(* Logix 5000 project; controller R1USB70001_CWRU_LOAD_20111116 vendor 1 type 14 code 54 rev 19.11; software revision 19.01 *)

TASK MainTask (continuous, watchdog 500 ms) : MainProgram

MODULES
   Local : vendor 1 type 14 code 54 (ICP 2, rev 19.11)
      CNB_LOAD : vendor 1 type 12 code 21 (ICP 0, rev 20.1)
         ACNR_RP_SC_N4 : vendor 1 type 12 code 111 (ControlNet 4, rev 1.1, Output RPI 8 ms)
            IE4C_RP_SC_S1 : 1734-IE4C (PointIO 1, rev 3.1, Input RPI 8 ms)
            IE4C_RP_SC_S2 : 1734-IE4C (PointIO 2, rev 3.1, Input RPI 8 ms)
            IE4C_RP_SC_S4 : 1734-IE4C (PointIO 4, rev 3.1, Input RPI 8 ms)
            IE4C_RP_SC_S3 : 1734-IE4C (PointIO 3, rev 3.1, Input RPI 8 ms)
            IE4C_RP_SC_S5 : 1734-IE4C (PointIO 5, rev 3.1, Input RPI 8 ms)
            IE4C_RP_SC_S6 : 1734-IE4C (PointIO 6, rev 3.1, Input RPI 8 ms)
            IE4C_RP_SC_S7 : 1734-IE4C (PointIO 7, rev 3.1, Input RPI 8 ms)
            IB8_RP_SC_S8 : 1734-IB8 (PointIO 8, rev 3.1)
            OB8_RP_SC_S10 : 1734-OB8 (PointIO 10, rev 3.1)
            OB8_RP_SC_S11 : 1734-OB8 (PointIO 11, rev 3.1)
            OB8_RP_SC_S12 : 1734-OB8 (PointIO 12, rev 3.1)
            OB8_RP_SC_S9 : 1734-OB8 (PointIO 9, rev 3.1)
         ACNR_CP_SC_N5 : vendor 1 type 12 code 111 (ControlNet 5, rev 1.1, Output RPI 8 ms)
            IE4C_CP_SC_S8 : 1734-IE4C (PointIO 8, rev 3.1, Input RPI 8 ms)
            IE4C_CP_SC_S1 : 1734-IE4C (PointIO 1, rev 3.1, Input RPI 8 ms)
            IE4C_CP_SC_S2 : 1734-IE4C (PointIO 2, rev 3.1, Input RPI 8 ms)
            IE4C_CP_SC_S3 : 1734-IE4C (PointIO 3, rev 3.1, Input RPI 8 ms)
            IE4C_CP_SC_S4 : 1734-IE4C (PointIO 4, rev 3.1, Input RPI 8 ms)
            IE4C_CP_SC_S6 : 1734-IE4C (PointIO 6, rev 3.1, Input RPI 8 ms)
            IE4C_CP_SC_S5 : 1734-IE4C (PointIO 5, rev 3.1, Input RPI 8 ms)
            IE4C_CP_SC_S7 : 1734-IE4C (PointIO 7, rev 3.1, Input RPI 8 ms)
            IB8_CP_SC_S9 : 1734-IB8 (PointIO 9, rev 3.1)
            OB8_CP_SC_S14 : 1734-OB8 (PointIO 13, rev 3.1)
            OB8_CP_SC_S13 : 1734-OB8 (PointIO 12, rev 3.1)
            OB8_CP_SC_S11 : 1734-OB8 (PointIO 10, rev 3.1)
            OB8_CP_SC_S12 : 1734-OB8 (PointIO 11, rev 3.1)
      EN2T_LOAD : 1756-EN2T (ICP 1, Ethernet 10.88.0.104, rev 4.3)
END_MODULES

VAR_GLOBAL   (* controller tags *)
   CL_LP_B1_ACAM : ALIAS FOR ACNR_CP_SC_N5:1:I.Ch1Data;
   CL_LP_B1_ACVS : ALIAS FOR ACNR_CP_SC_N5:9:I.1;
   CL_LP_B1_L1_ACAM : ALIAS FOR ACNR_CP_SC_N5:1:I.Ch2Data;
   CL_LP_B1_L2_ACAM : ALIAS FOR ACNR_CP_SC_N5:1:I.Ch3Data;
   CL_LP_B1_L3_ACAM : ALIAS FOR ACNR_CP_SC_N5:2:I.Ch0Data;
   CL_LP_B1_L4_ACAM : ALIAS FOR ACNR_CP_SC_N5:2:I.Ch1Data;
   CL_LP_B1_L5_ACAM : ALIAS FOR ACNR_CP_SC_N5:2:I.Ch2Data;
   CL_LP_B2_ACAM : ALIAS FOR ACNR_CP_SC_N5:2:I.Ch3Data;
   CL_LP_B2_ACVS : ALIAS FOR ACNR_CP_SC_N5:9:I.2;
   CL_LP_B2_L1_ACAM : ALIAS FOR ACNR_CP_SC_N5:3:I.Ch0Data;
   CL_LP_B2_L2_ACAM : ALIAS FOR ACNR_CP_SC_N5:3:I.Ch1Data;
   CL_LP_B2_L3_ACAM : ALIAS FOR ACNR_CP_SC_N5:3:I.Ch2Data;
   CL_LP_B2_L4_ACAM : ALIAS FOR ACNR_CP_SC_N5:3:I.Ch3Data;
   CL_LP_B2_L5_ACAM : ALIAS FOR ACNR_CP_SC_N5:4:I.Ch0Data;
   CL_LP_ML_ACAM : ALIAS FOR ACNR_CP_SC_N5:1:I.Ch0Data;
   CL_LP_ML_ACVT : ALIAS FOR ACNR_CP_SC_N5:7:I.Ch2Data;
   CL_TIMER00 : TIMER;
   COM_B1_Alias : ALIAS FOR ACNR_CP_SC_N5:10:O.1;
   COM_B1_LOAD1_Alias : ALIAS FOR ACNR_CP_SC_N5:10:O.2;
   COM_B1_LOAD1_USER : BOOL;
   COM_B1_LOAD2_Alias : ALIAS FOR ACNR_CP_SC_N5:10:O.3;
   COM_B1_LOAD2_USER : BOOL;
   COM_B1_LOAD3_Alias : ALIAS FOR ACNR_CP_SC_N5:10:O.4;
   COM_B1_LOAD3_USER : BOOL;
   COM_B1_LOAD4_Alias : ALIAS FOR ACNR_CP_SC_N5:10:O.5;
   COM_B1_LOAD4_USER : BOOL;
   COM_B1_LOAD5_Alias : ALIAS FOR ACNR_CP_SC_N5:10:O.6;
   COM_B1_LOAD5_USER : BOOL;
   COM_B1_USER : BOOL;
   COM_B2_Alias : ALIAS FOR ACNR_CP_SC_N5:10:O.7;
   COM_B2_LOAD1_Alias : ALIAS FOR ACNR_CP_SC_N5:11:O.0;
   COM_B2_LOAD1_USER : BOOL;
   COM_B2_LOAD2_Alias : ALIAS FOR ACNR_CP_SC_N5:11:O.1;
   COM_B2_LOAD2_USER : BOOL;
   COM_B2_LOAD3_Alias : ALIAS FOR ACNR_CP_SC_N5:11:O.2;
   COM_B2_LOAD3_USER : BOOL;
   COM_B2_LOAD4_Alias : ALIAS FOR ACNR_CP_SC_N5:11:O.3;
   COM_B2_LOAD4_USER : BOOL;
   COM_B2_LOAD5_Alias : ALIAS FOR ACNR_CP_SC_N5:11:O.4;
   COM_B2_LOAD5_USER : BOOL;
   COM_B2_USER : BOOL;
   COM_MAIN_Alias : ALIAS FOR ACNR_CP_SC_N5:10:O.0;
   COM_MAIN_CLOSE : BOOL;
   COM_MAIN_CLOSE_Alias : BOOL;
   COM_MAIN_USER : BOOL;
   Comment : DINT[2] := ([0] := 3);
   HMI_Intfc_Read_Buffer : DINT[66] := ([0] := 235, [1] := 560, [2] := 5614, [3] := -31, [4] := -66, [5] := -101, [6] := 317, [7] := -1, [8] := 114, [9] := 102, [10] := 69, [11] := -7, [12] := 37, [13] := -1, [14] := 64, [15] := 82, [16] := -48, [17] := 42, [18] := 138, [20] := 25, [21] := 35, [22] := -29, [23] := 66, [25] := 7, [26] := -17, [27] := -13, [28] := 22, [29] := 1048839, [30] := 430, [31] := 431, [34] := 97, [35] := -66, [36] := -44, [37] := 52, [38] := 59, [40] := 5, [41] := 5, [42] := 68, [43] := 24, [44] := -84, [46] := -1, [47] := 56, [48] := -6, [49] := 66, [50] := 126, [51] := 109, [53] := 64, [54] := 77, [55] := 6, [56] := 31, [57] := 37, [59] := 1, [60] := 3294, [61] := -16, [62] := -15, [63] := -12);
        [0]   // RL_LP_ML_ACAM
        [1]   // RL_LP_B1_ACAM
        [2]   // RL_LP_B1_L1_ACAM
        [3]   // RL_LP_B1_L2_ACAM
        [4]   // RL_LP_B1_L3_ACAM
        [5]   // RL_LP_B1_L4_ACAM
        [6]   // RL_LP_B1_L5_ACAM
        [7]   // RL_LP_B2_ACAM
        [8]   // RL_LP_B2_L1_ACAM
        [9]   // RL_LP_B2_L2_ACAM
        [10]   // RL_LP_B2_L3_ACAM
        [11]   // RL_LP_B2_L4_ACAM
        [26]   // SPARE RESERVED FOR SLOT 7 CHANNEL 2
        [27]   // SPARE RESERVED FOR SLOT 7 CHANNEL 3
        [63]   // SPARE RESERVED FOR SLOT 8 CHANNEL 3
        [62]   // SPARE RESERVED FOR SLOT 8 CHANNEL 2
        [61]   // SPARE RESERVED FOR SLOT 8 CHANNEL 1
        [60]   // SPARE RESERVED FOR SLOT 8 CHANNEL 0
        [12]   // RL_LP_B2_L5_ACAM
        [13]   // RL_LP_B3_ACAM
        [14]   // RL_LP_B3_L1_ACAM
        [15]   // RL_LP_B3_L2_ACAM
        [16]   // RL_LP_B3_L3_ACAM
        [17]   // RL_LP_B3_L4_ACAM
        [18]   // RL_LP_B3_L5_ACAM
        [19]   // RL_LP_B4_ACAM
        [20]   // RL_LP_B4_L1_ACAM
        [21]   // RL_LP_B4_L2_ACAM
        [22]   // RL_LP_B4_L3_ACAM
        [23]   // RL_LP_B4_L4_ACAM
        [24]   // RL_LP_B4_L5_ACAM
        [25]   // RL_LP_ML_ACVT
        [28].1   // RL_LP_B1_ACVS
        [28].2   // RL_LP_B2_ACVS
        [28].3   // RL_LP_B3_ACVS
        [28].4   // RL_LP_B4_ACVS
        [29].0   // RL_LP_ML_CS
        [29].1   // RL_LP_B1_CS
        [29].2   // RL_LP_B1_L1_CS
        [29].3   // RL_LP_B1_L2_CS
        [29].4   // RL_LP_B1_L3_CS
        [29].5   // RL_LP_B1_L4_CS
        [29].6   // RL_LP_B1_L5_CS
        [29].8   // RL_LP_B2_CS
        [29].9   // RL_LP_B2_L1_CS
        [29].10   // RL_LP_B2_L2_CS
        [29].11   // RL_LP_B2_L3_CS
        [29].12   // RL_LP_B2_L4_CS
        [29].13   // RL_LP_B2_L5_CS
        [29].14   // RL_LP_B3_CS
        [29].15   // RL_LP_B3_L1_CS
        [29].16   // RL_LP_B3_L2_CS
        [29].17   // RL_LP_B3_L3_CS
        [29].18   // RL_LP_B3_L4_CS
        [29].19   // RL_LP_B3_L5_CS
        [29].20   // RL_LP_B4_CS
        [29].21   // RL_LP_B4_L1_CS
        [29].22   // RL_LP_B4_L2_CS
        [29].23   // RL_LP_B4_L3_CS
        [29].24   // RL_LP_B4_L4_CS
        [29].25   // RL_LP_B4_L5_CS
        [32]   // CL_LP_ML_ACAM
        [33]   // CL_LP_B1_ACAM
        [34]   // CL_LP_B1_L1_ACAM
        [35]   // CL_LP_B1_L2_ACAM
        [36]   // CL_LP_B1_L3_ACAM
        [37]   // CL_LP_B1_L4_ACAM
        [38]   // CL_LP_B1_L5_ACAM
        [39]   // CL_LP_B2_ACAM
        [40]   // CL_LP_B2_L1_ACAM
        [41]   // CL_LP_B2_L2_ACAM
        [42]   // CL_LP_B2_L3_ACAM
        [43]   // CL_LP_B2_L4_ACAM
        [44]   // CL_LP_B2_L5_ACAM
        [45]   // IL_LP_ML_ACAM
        [46]   // IL_LP_B1_ACAM
        [47]   // IL_LP_B1_L1_ACAM
        [48]   // IL_LP_B1_L2_ACAM
        [49]   // IL_LP_B1_L3_ACAM
        [50]   // IL_LP_B1_L4_ACAM
        [51]   // IL_LP_B1_L5_ACAM
        [52]   // IL_LP_B2_ACAM
        [53]   // IL_LP_B2_L1_ACAM
        [54]   // IL_LP_B2_L2_ACAM
        [55]   // IL_LP_B2_L3_ACAM
        [56]   // IL_LP_B2_L4_ACAM
        [57]   // IL_LP_B2_L5_ACAM
        [58]   // CL_LP_ML_ACVT
        [59]   // IL_LP_ML_ACVT
        [64].1   // CL_LP_B1_ACVS
        [64].2   // CL_LP_B2_ACVS
        [64].4   // IL_LP_B1_ACVS
        [64].5   // IL_LP_B2_ACVS
        [65].0   // CL_LP_ML_CS
        [65].1   // CL_LP_B1_CS
        [65].2   // CL_LP_B1_L1_CS
        [65].3   // CL_LP_B1_L2_CS
        [65].4   // CL_LP_B1_L3_CS
        [65].5   // CL_LP_B1_L4_CS
        [65].6   // CL_LP_B1_L5_CS
        [65].7   // CL_LP_B2_CS
        [65].8   // CL_LP_B2_L1_CS
        [65].9   // CL_LP_B2_L2_CS
        [65].10   // CL_LP_B2_L3_CS
        [65].11   // CL_LP_B2_L4_CS
        [65].12   // CL_LP_B2_L5_CS
        [65].13   // IL_LP_ML_CS
        [65].14   // IL_LP_B1_CS
        [65].15   // IL_LP_B1_L1_CS
        [65].16   // IL_LP_B1_L2_CS
        [65].17   // IL_LP_B1_L3_CS
        [65].18   // IL_LP_B1_L4_CS
        [65].19   // IL_LP_B1_L5_CS
        [65].20   // IL_LP_B2_CS
        [65].21   // IL_LP_B2_L1_CS
        [65].22   // IL_LP_B2_L2_CS
        [65].23   // IL_LP_B2_L3_CS
        [65].24   // IL_LP_B2_L4_CS
        [65].25   // IL_LP_B2_L5_CS
   IL_LP_B1_ACAM : ALIAS FOR ACNR_CP_SC_N5:4:I.Ch2Data;
   IL_LP_B1_ACVS : ALIAS FOR ACNR_CP_SC_N5:9:I.4;
   IL_LP_B1_L1_ACAM : ALIAS FOR ACNR_CP_SC_N5:4:I.Ch3Data;
   IL_LP_B1_L2_ACAM : ALIAS FOR ACNR_CP_SC_N5:5:I.Ch0Data;
   IL_LP_B1_L3_ACAM : ALIAS FOR ACNR_CP_SC_N5:5:I.Ch1Data;
   IL_LP_B1_L4_ACAM : ALIAS FOR ACNR_CP_SC_N5:5:I.Ch2Data;
   IL_LP_B1_L5_ACAM : ALIAS FOR ACNR_CP_SC_N5:5:I.Ch3Data;
   IL_LP_B2_ACAM : ALIAS FOR ACNR_CP_SC_N5:6:I.Ch0Data;
   IL_LP_B2_ACVS : ALIAS FOR ACNR_CP_SC_N5:9:I.5;
   IL_LP_B2_L1_ACAM : ALIAS FOR ACNR_CP_SC_N5:6:I.Ch1Data;
   IL_LP_B2_L2_ACAM : ALIAS FOR ACNR_CP_SC_N5:6:I.Ch2Data;
   IL_LP_B2_L3_ACAM : ALIAS FOR ACNR_CP_SC_N5:6:I.Ch3Data;
   IL_LP_B2_L4_ACAM : ALIAS FOR ACNR_CP_SC_N5:7:I.Ch0Data;
   IL_LP_B2_L5_ACAM : ALIAS FOR ACNR_CP_SC_N5:7:I.Ch1Data;
   IL_LP_ML_ACAM : ALIAS FOR ACNR_CP_SC_N5:4:I.Ch1Data;
   IL_LP_ML_ACVT : ALIAS FOR ACNR_CP_SC_N5:7:I.Ch3Data;
   IND_B1_Alias : ALIAS FOR ACNR_CP_SC_N5:11:O.6;
   IND_B1_LOAD1_Alias : ALIAS FOR ACNR_CP_SC_N5:11:O.7;
   IND_B1_LOAD1_USER : BOOL;
   IND_B1_LOAD2_Alias : ALIAS FOR ACNR_CP_SC_N5:12:O.0;
   IND_B1_LOAD2_USER : BOOL;
   IND_B1_LOAD3_Alias : ALIAS FOR ACNR_CP_SC_N5:12:O.1;
   IND_B1_LOAD3_USER : BOOL;
   IND_B1_LOAD4_Alias : ALIAS FOR ACNR_CP_SC_N5:12:O.2;
   IND_B1_LOAD4_USER : BOOL;
   IND_B1_LOAD5_Alias : ALIAS FOR ACNR_CP_SC_N5:12:O.3;
   IND_B1_LOAD5_USER : BOOL;
   IND_B1_USER : BOOL;
   IND_B2_Alias : ALIAS FOR ACNR_CP_SC_N5:12:O.4;
   IND_B2_LOAD1_Alias : ALIAS FOR ACNR_CP_SC_N5:12:O.5;
   IND_B2_LOAD1_USER : BOOL;
   IND_B2_LOAD2_Alias : ALIAS FOR ACNR_CP_SC_N5:12:O.6;
   IND_B2_LOAD2_USER : BOOL;
   IND_B2_LOAD3_Alias : ALIAS FOR ACNR_CP_SC_N5:12:O.7;
   IND_B2_LOAD3_USER : BOOL;
   IND_B2_LOAD4_Alias : ALIAS FOR ACNR_CP_SC_N5:13:O.0;
   IND_B2_LOAD4_USER : BOOL;
   IND_B2_LOAD5_Alias : ALIAS FOR ACNR_CP_SC_N5:13:O.1;
   IND_B2_LOAD5_USER : BOOL;
   IND_B2_USER : BOOL;
   IND_MAIN_Alias : ALIAS FOR ACNR_CP_SC_N5:11:O.5;
   IND_MAIN_USER : BOOL;
   RES_B1_Alias : ALIAS FOR ACNR_RP_SC_N4:9:O.1;
   RES_B1_LOAD1_Alias : ALIAS FOR ACNR_RP_SC_N4:9:O.2;
   RES_B1_LOAD1_USER : BOOL;
   RES_B1_LOAD2_Alias : ALIAS FOR ACNR_RP_SC_N4:9:O.3;
   RES_B1_LOAD2_USER : BOOL;
   RES_B1_LOAD3_Alias : ALIAS FOR ACNR_RP_SC_N4:9:O.4;
   RES_B1_LOAD3_USER : BOOL;
   RES_B1_LOAD4_Alias : ALIAS FOR ACNR_RP_SC_N4:9:O.5;
   RES_B1_LOAD4_USER : BOOL;
   RES_B1_LOAD5_Alias : ALIAS FOR ACNR_RP_SC_N4:9:O.6;
   RES_B1_LOAD5_USER : BOOL;
   RES_B1_USER : BOOL;
   RES_B2_Alias : ALIAS FOR ACNR_RP_SC_N4:10:O.0;
   RES_B2_LOAD1_Alias : ALIAS FOR ACNR_RP_SC_N4:10:O.1;
   RES_B2_LOAD1_USER : BOOL;
   RES_B2_LOAD2_Alias : ALIAS FOR ACNR_RP_SC_N4:10:O.2;
   RES_B2_LOAD2_USER : BOOL;
   RES_B2_LOAD3_Alias : ALIAS FOR ACNR_RP_SC_N4:10:O.3;
   RES_B2_LOAD3_USER : BOOL;
   RES_B2_LOAD4_Alias : ALIAS FOR ACNR_RP_SC_N4:10:O.4;
   RES_B2_LOAD4_USER : BOOL;
   RES_B2_LOAD5_Alias : ALIAS FOR ACNR_RP_SC_N4:10:O.5;
   RES_B2_LOAD5_USER : BOOL;
   RES_B2_USER : BOOL;
   RES_B3_Alias : ALIAS FOR ACNR_RP_SC_N4:10:O.6;
   RES_B3_LOAD1_Alias : ALIAS FOR ACNR_RP_SC_N4:10:O.7;
   RES_B3_LOAD1_USER : BOOL;
   RES_B3_LOAD2_Alias : ALIAS FOR ACNR_RP_SC_N4:11:O.0;
   RES_B3_LOAD2_USER : BOOL;
   RES_B3_LOAD3_Alias : ALIAS FOR ACNR_RP_SC_N4:11:O.1;
   RES_B3_LOAD3_USER : BOOL;
   RES_B3_LOAD4_Alias : ALIAS FOR ACNR_RP_SC_N4:11:O.2;
   RES_B3_LOAD4_USER : BOOL;
   RES_B3_LOAD5_Alias : ALIAS FOR ACNR_RP_SC_N4:11:O.3;
   RES_B3_LOAD5_USER : BOOL;
   RES_B3_USER : BOOL;
   RES_B4_Alias : ALIAS FOR ACNR_RP_SC_N4:11:O.4;
   RES_B4_LOAD1_Alias : ALIAS FOR ACNR_RP_SC_N4:11:O.5;
   RES_B4_LOAD1_USER : BOOL;
   RES_B4_LOAD2_Alias : ALIAS FOR ACNR_RP_SC_N4:11:O.6;
   RES_B4_LOAD2_USER : BOOL;
   RES_B4_LOAD3_Alias : ALIAS FOR ACNR_RP_SC_N4:11:O.7;
   RES_B4_LOAD3_USER : BOOL;
   RES_B4_LOAD4_Alias : ALIAS FOR ACNR_RP_SC_N4:12:O.0;
   RES_B4_LOAD4_USER : BOOL;
   RES_B4_LOAD5_Alias : ALIAS FOR ACNR_RP_SC_N4:12:O.1;
   RES_B4_LOAD5_USER : BOOL;
   RES_B4_USER : BOOL;
   RES_MAIN_Alias : ALIAS FOR ACNR_RP_SC_N4:9:O.0;
   RES_MAIN_USER : BOOL;
   RESB1_LOAD1_USER : BOOL;
   RESB2_LOAD2_USER : BOOL;
   RL_LP_B1_ACAM : ALIAS FOR ACNR_RP_SC_N4:1:I.Ch1Data;
   RL_LP_B1_ACVS : ALIAS FOR ACNR_RP_SC_N4:8:I.1;
   RL_LP_B1_L1_ACAM : ALIAS FOR ACNR_RP_SC_N4:1:I.Ch2Data;
   RL_LP_B1_L2_ACAM : ALIAS FOR ACNR_RP_SC_N4:1:I.Ch3Data;
   RL_LP_B1_L3_ACAM : ALIAS FOR ACNR_RP_SC_N4:2:I.Ch0Data;
   RL_LP_B1_L4_ACAM : ALIAS FOR ACNR_RP_SC_N4:2:I.Ch1Data;
   RL_LP_B1_L5_ACAM : ALIAS FOR ACNR_RP_SC_N4:2:I.Ch2Data;
   RL_LP_B2_ACAM : ALIAS FOR ACNR_RP_SC_N4:2:I.Ch3Data;
   RL_LP_B2_ACVS : ALIAS FOR ACNR_RP_SC_N4:8:I.2;
   RL_LP_B2_L1_ACAM : ALIAS FOR ACNR_RP_SC_N4:3:I.Ch0Data;
   RL_LP_B2_L2_ACAM : ALIAS FOR ACNR_RP_SC_N4:3:I.Ch1Data;
   RL_LP_B2_L3_ACAM : ALIAS FOR ACNR_RP_SC_N4:3:I.Ch2Data;
   RL_LP_B2_L4_ACAM : ALIAS FOR ACNR_RP_SC_N4:3:I.Ch3Data;
   RL_LP_B2_L5_ACAM : ALIAS FOR ACNR_RP_SC_N4:4:I.Ch0Data;
   RL_LP_B3_ACAM : ALIAS FOR ACNR_RP_SC_N4:4:I.Ch1Data;
   RL_LP_B3_ACVS : ALIAS FOR ACNR_RP_SC_N4:8:I.3;
   RL_LP_B3_L1_ACAM : ALIAS FOR ACNR_RP_SC_N4:4:I.Ch2Data;
   RL_LP_B3_L2_ACAM : ALIAS FOR ACNR_RP_SC_N4:4:I.Ch3Data;
   RL_LP_B3_L3_ACAM : ALIAS FOR ACNR_RP_SC_N4:5:I.Ch0Data;
   RL_LP_B3_L4_ACAM : ALIAS FOR ACNR_RP_SC_N4:5:I.Ch1Data;
   RL_LP_B3_L5_ACAM : ALIAS FOR ACNR_RP_SC_N4:5:I.Ch2Data;
   RL_LP_B4_ACAM : ALIAS FOR ACNR_RP_SC_N4:5:I.Ch3Data;
   RL_LP_B4_ACVS : ALIAS FOR ACNR_RP_SC_N4:8:I.4;
   RL_LP_B4_L1_ACAM : ALIAS FOR ACNR_RP_SC_N4:6:I.Ch0Data;
   RL_LP_B4_L2_ACAM : ALIAS FOR ACNR_RP_SC_N4:6:I.Ch1Data;
   RL_LP_B4_L3_ACAM : ALIAS FOR ACNR_RP_SC_N4:6:I.Ch2Data;
   RL_LP_B4_L4_ACAM : ALIAS FOR ACNR_RP_SC_N4:6:I.Ch3Data;
   RL_LP_B4_L5_ACAM : ALIAS FOR ACNR_RP_SC_N4:7:I.Ch0Data;
   RL_LP_ML_ACAM : ALIAS FOR ACNR_RP_SC_N4:1:I.Ch0Data;
   RL_LP_ML_ACVT : ALIAS FOR ACNR_RP_SC_N4:7:I.Ch1Data;
END_VAR

PROGRAM MainProgram   (* main routine MainRoutine *)
VAR
   COM_B1_CLOSE_PROXY : BOOL;
   COM_B1_CLOSED : BOOL;
   COM_B1_COMMAND_CHANGED : BOOL;
   COM_B1_COMMAND_CHANGED_TIMER : TIMER;
   COM_B1_CURRENT_CHECK : REAL := 0.0059203943;
   COM_B1_CURRENT_RAW : REAL;
   COM_B1_DISCREPANCY : REAL := 0.0059203943;
   COM_B1_FAULT_CANCEL : BOOL := 1;
   COM_B1_FAULT_PENDING : BOOL;
   COM_B1_FAULT_REQ : BOOL;
   COM_B1_FAULT_RETHROW_TIMER : TIMER := (PRE := 100);
   COM_B1_FAULT_TRIP : BOOL;
   COM_B1_INT_REQ_CLOSE : BOOL;
   COM_B1_INT_REQ_CONNECT : BOOL;
   COM_B1_MISMATCH : BOOL;
   COM_B1_NEW_FAULT : BOOL;
   COM_B1_RECLOSE_COUNTER : DINT;
   COM_B1_RECLOSE_OFF : BOOL;
   COM_B1_RECLOSE_TIMER : TIMER := (PRE := 1000);
   COM_B1_RECLOSED : BOOL;
   COM_B1_REQ_CLOSE : BOOL;
   COM_B1_REQ_CONNECT : BOOL;
   COM_B1_REQ_DISCONNECT : BOOL;
   COM_B1_REQ_OPEN : BOOL := 1;
   COM_B1_REQ_RECLOSE : BOOL;
   COM_B1_SENSOR_ERROR : BOOL;
   COM_B1L1_CURRENT : REAL := 0.005920395;
   COM_B1L1_CURRENT_RAW : REAL := 97.0;
   COM_B1L2_CURRENT : REAL := -0.00402831;
   COM_B1L2_CURRENT_RAW : REAL := -66.0;
   COM_B1L3_CURRENT : REAL := -0.002746575;
   COM_B1L3_CURRENT_RAW : REAL := -45.0;
   COM_B1L4_CURRENT : REAL := 0.00317382;
   COM_B1L4_CURRENT_RAW : REAL := 52.0;
   COM_B1L5_CURRENT : REAL := 0.003601065;
   COM_B1L5_CURRENT_RAW : REAL := 59.0;
   COM_B2_CLOSE_PROXY : BOOL;
   COM_B2_CLOSED : BOOL;
   COM_B2_COMMAND_CHANGED : BOOL;
   COM_B2_COMMAND_CHANGED_TIMER : TIMER;
   COM_B2_CURRENT_CHECK : REAL := 0.00109863;
   COM_B2_CURRENT_RAW : REAL;
   COM_B2_DISCREPANCY : REAL := 0.00109863;
   COM_B2_FAULT_CANCEL : BOOL := 1;
   COM_B2_FAULT_PENDING : BOOL;
   COM_B2_FAULT_REQ : BOOL;
   COM_B2_FAULT_RETHROW_TIMER : TIMER := (PRE := 100);
   COM_B2_FAULT_TRIP : BOOL;
   COM_B2_INT_REQ_CLOSE : BOOL;
   COM_B2_INT_REQ_CONNECT : BOOL;
   COM_B2_MISMATCH : BOOL;
   COM_B2_NEW_FAULT : BOOL;
   COM_B2_RECLOSE_COUNTER : DINT;
   COM_B2_RECLOSE_OFF : BOOL;
   COM_B2_RECLOSE_TIMER : TIMER := (PRE := 1000);
   COM_B2_RECLOSED : BOOL;
   COM_B2_REQ_CLOSE : BOOL;
   COM_B2_REQ_CONNECT : BOOL;
   COM_B2_REQ_DISCONNECT : BOOL;
   COM_B2_REQ_OPEN : BOOL := 1;
   COM_B2_REQ_RECLOSE : BOOL;
   COM_B2_SENSOR_ERROR : BOOL;
   COM_B2L1_CURRENT : REAL := 0.000305175;
   COM_B2L1_CURRENT_RAW : REAL := 5.0;
   COM_B2L2_CURRENT : REAL := 0.000305175;
   COM_B2L2_CURRENT_RAW : REAL := 5.0;
   COM_B2L3_CURRENT : REAL := 0.00415038;
   COM_B2L3_CURRENT_RAW : REAL := 68.0;
   COM_B2L4_CURRENT : REAL := 0.00146484;
   COM_B2L4_CURRENT_RAW : REAL := 24.0;
   COM_B2L5_CURRENT : REAL := -0.00512694;
   COM_B2L5_CURRENT_RAW : REAL := -84.0;
   COM_BUS1_CURRENT : REAL;
   COM_BUS2_CURRENT : REAL;
   COM_BUS_FAULT_THRESHOLD : REAL := 2.0;
   COM_HighVoltage : BOOL;
   COM_HighVoltageThreshold : REAL;
   COM_LowVoltage : BOOL;
   COM_LowVoltageThreshold : REAL;
   COM_MAIN_CLOSE_PROXY : BOOL;
   COM_MAIN_CLOSED : BOOL;
   COM_MAIN_COMMAND_CHANGED : BOOL;
   COM_MAIN_COMMAND_CHANGED_TIMER : TIMER;
   COM_MAIN_CURRENT : REAL;
   COM_MAIN_CURRENT_CHECK : REAL;
   COM_MAIN_CURRENT_RAW : REAL;
   COM_MAIN_DISCREPANCY : REAL;
   COM_MAIN_FAULT_CANCEL : BOOL;
   COM_MAIN_FAULT_PENDING : BOOL := 1;
   COM_MAIN_FAULT_REQ : BOOL := 1;
   COM_MAIN_FAULT_RETHROW_TIMER : TIMER := (PRE := 100);
   COM_MAIN_FAULT_THRESHOLD : REAL;
   COM_MAIN_FAULT_TRIP : BOOL := 1;
   COM_MAIN_INT_REQ_CLOSE : BOOL;
   COM_MAIN_INT_REQ_CONNECT : BOOL;
   COM_MAIN_MISMATCH : BOOL := 1;
   COM_MAIN_NEW_FAULT : BOOL;
   COM_MAIN_RECLOSE_COUNTER : DINT := 75;
   COM_MAIN_RECLOSE_OFF : BOOL := 1;
   COM_MAIN_RECLOSE_TIMER : TIMER := (PRE := 1000);
   COM_MAIN_RECLOSED : BOOL;
   COM_MAIN_REQ_CLOSE : BOOL;
   COM_MAIN_REQ_CONNECT : BOOL;
   COM_MAIN_REQ_DISCONNECT : BOOL;
   COM_MAIN_REQ_OPEN : BOOL := 1;
   COM_MAIN_REQ_RECLOSE : BOOL;
   COM_MAIN_SENSOR_ERROR : BOOL;
   COM_MAIN_VOLTAGE : REAL;
   COM_MAIN_VOLTAGE_RAW : REAL;
   CURRENT_SCALE_HIGH : REAL := 0.00061037;
   CURRENT_SCALE_LOW : REAL := 6.1035e-05;
   IND_B1_CLOSE_PROXY : BOOL;
   IND_B1_CLOSED : BOOL;
   IND_B1_COMMAND_CHANGED : BOOL;
   IND_B1_COMMAND_CHANGED_TIMER : TIMER;
   IND_B1_CURRENT_CHECK : REAL := 0.021423286;
   IND_B1_CURRENT_RAW : REAL := -1.0;
   IND_B1_DISCREPANCY : REAL := 0.022033656;
   IND_B1_FAULT_CANCEL : BOOL;
   IND_B1_FAULT_PENDING : BOOL := 1;
   IND_B1_FAULT_REQ : BOOL := 1;
   IND_B1_FAULT_RETHROW_TIMER : TIMER := (PRE := 100);
   IND_B1_FAULT_TRIP : BOOL := 1;
   IND_B1_INT_REQ_CLOSE : BOOL;
   IND_B1_INT_REQ_CONNECT : BOOL;
   IND_B1_MISMATCH : BOOL := 1;
   IND_B1_NEW_FAULT : BOOL;
   IND_B1_RECLOSE_COUNTER : DINT := 75;
   IND_B1_RECLOSE_OFF : BOOL := 1;
   IND_B1_RECLOSE_TIMER : TIMER := (PRE := 1000);
   IND_B1_RECLOSED : BOOL;
   IND_B1_REQ_CLOSE : BOOL;
   IND_B1_REQ_CONNECT : BOOL;
   IND_B1_REQ_DISCONNECT : BOOL;
   IND_B1_REQ_OPEN : BOOL := 1;
   IND_B1_REQ_RECLOSE : BOOL;
   IND_B1_SENSOR_ERROR : BOOL;
   IND_B1L1_CURRENT : REAL := 0.003478995;
   IND_B1L1_CURRENT_RAW : REAL := 57.0;
   IND_B1L2_CURRENT : REAL := -0.00036621;
   IND_B1L2_CURRENT_RAW : REAL := -6.0;
   IND_B1L3_CURRENT : REAL := 0.00402831;
   IND_B1L3_CURRENT_RAW : REAL := 66.0;
   IND_B1L4_CURRENT : REAL := 0.00769041;
   IND_B1L4_CURRENT_RAW : REAL := 126.0;
   IND_B1L5_CURRENT : REAL := 0.00659178;
   IND_B1L5_CURRENT_RAW : REAL := 108.0;
   IND_B2_CLOSE_PROXY : BOOL;
   IND_B2_CLOSED : BOOL;
   IND_B2_COMMAND_CHANGED : BOOL;
   IND_B2_COMMAND_CHANGED_TIMER : TIMER;
   IND_B2_CURRENT_CHECK : REAL := 0.01318356;
   IND_B2_CURRENT_RAW : REAL := -1.0;
   IND_B2_DISCREPANCY : REAL := 0.01379393;
   IND_B2_FAULT_CANCEL : BOOL;
   IND_B2_FAULT_PENDING : BOOL := 1;
   IND_B2_FAULT_REQ : BOOL := 1;
   IND_B2_FAULT_RETHROW_TIMER : TIMER := (PRE := 100);
   IND_B2_FAULT_TRIP : BOOL := 1;
   IND_B2_INT_REQ_CLOSE : BOOL;
   IND_B2_INT_REQ_CONNECT : BOOL;
   IND_B2_MISMATCH : BOOL := 1;
   IND_B2_NEW_FAULT : BOOL;
   IND_B2_RECLOSE_COUNTER : DINT := 75;
   IND_B2_RECLOSE_OFF : BOOL := 1;
   IND_B2_RECLOSE_TIMER : TIMER := (PRE := 1000);
   IND_B2_RECLOSED : BOOL;
   IND_B2_REQ_CLOSE : BOOL;
   IND_B2_REQ_CONNECT : BOOL;
   IND_B2_REQ_DISCONNECT : BOOL;
   IND_B2_REQ_OPEN : BOOL := 1;
   IND_B2_REQ_RECLOSE : BOOL;
   IND_B2_SENSOR_ERROR : BOOL;
   IND_B2L1_CURRENT : REAL := 0.00402831;
   IND_B2L1_CURRENT_RAW : REAL := 65.0;
   IND_B2L2_CURRENT : REAL := 0.004699695;
   IND_B2L2_CURRENT_RAW : REAL := 77.0;
   IND_B2L3_CURRENT : REAL := 0.00036621;
   IND_B2L3_CURRENT_RAW : REAL := 6.0;
   IND_B2L4_CURRENT : REAL := 0.001892085;
   IND_B2L4_CURRENT_RAW : REAL := 31.0;
   IND_B2L5_CURRENT : REAL := 0.002258295;
   IND_B2L5_CURRENT_RAW : REAL := 37.0;
   IND_BUS1_CURRENT : REAL := -0.00061037;
   IND_BUS2_CURRENT : REAL := -0.00061037;
   IND_BUS_FAULT_THRESHOLD : REAL;
   IND_HighVoltage : BOOL;
   IND_LowVoltage : BOOL;
   IND_LowVoltageThreshold : REAL;
   IND_MAIN_CLOSE_PROXY : BOOL;
   IND_MAIN_CLOSED : BOOL;
   IND_MAIN_COMMAND_CHANGED : BOOL;
   IND_MAIN_COMMAND_CHANGED_TIMER : TIMER;
   IND_MAIN_CURRENT : REAL;
   IND_MAIN_CURRENT_CHECK : REAL := -0.00122074;
   IND_MAIN_CURRENT_RAW : REAL;
   IND_MAIN_DISCREPANCY : REAL := 0.00122074;
   IND_MAIN_FAULT_CANCEL : BOOL;
   IND_MAIN_FAULT_PENDING : BOOL := 1;
   IND_MAIN_FAULT_REQ : BOOL := 1;
   IND_MAIN_FAULT_RETHROW_TIMER : TIMER := (PRE := 100);
   IND_MAIN_FAULT_THRESHOLD : REAL;
   IND_MAIN_FAULT_TRIP : BOOL := 1;
   IND_MAIN_INT_REQ_CLOSE : BOOL;
   IND_MAIN_INT_REQ_CONNECT : BOOL;
   IND_MAIN_MISMATCH : BOOL := 1;
   IND_MAIN_NEW_FAULT : BOOL;
   IND_MAIN_RECLOSE_COUNTER : DINT := 75;
   IND_MAIN_RECLOSE_OFF : BOOL := 1;
   IND_MAIN_RECLOSE_TIMER : TIMER := (PRE := 1000);
   IND_MAIN_RECLOSED : BOOL;
   IND_MAIN_REQ_CLOSE : BOOL;
   IND_MAIN_REQ_CONNECT : BOOL;
   IND_MAIN_REQ_DISCONNECT : BOOL;
   IND_MAIN_REQ_OPEN : BOOL := 1;
   IND_MAIN_REQ_RECLOSE : BOOL;
   IND_MAIN_SENSOR_ERROR : BOOL;
   IND_MAIN_VOLTAGE : REAL;
   IND_MAIN_VOLTAGE_RAW : REAL;
   INITIALIZATION_GUARD : BOOL;
   INITIALIZATION_GUARD_INT : BOOL;
   INITIALIZE_GRID : BOOL;
   OkToConnect : BOOL;
   RECLOSE_LIMIT : DINT := 4;
   RES_B1_CLOSE_PROXY : BOOL := 1;
   RES_B1_CLOSED : BOOL := 1;
   RES_B1_COMMAND_CHANGED : BOOL;
   RES_B1_COMMAND_CHANGED_TIMER : TIMER;
   RES_B1_CURRENT_CHECK : REAL := 0.35388094;
   RES_B1_CURRENT_RAW : REAL := 561.0;
   RES_B1_DISCREPANCY : REAL := 0.011463374;
   RES_B1_FAULT : BOOL;
   RES_B1_FAULT_CANCEL : BOOL := 1;
   RES_B1_FAULT_PENDING : BOOL;
   RES_B1_FAULT_REQ : BOOL;
   RES_B1_FAULT_RETHROW_TIMER : TIMER := (PRE := 100);
   RES_B1_FAULT_TRIP : BOOL;
   RES_B1_INT_REQ_CLOSE : BOOL := 1;
   RES_B1_INT_REQ_CONNECT : BOOL := 1;
   RES_B1_MATCH_TIMER : TIMER := (PRE := 25, ACC := 25, EN := 1, DN := 1);
   RES_B1_MISMATCH : BOOL;
   RES_B1_MISMATCH_TIMER : TIMER := (PRE := 25);
   RES_B1_NEW_FAULT : BOOL;
   RES_B1_RECLOSE_COUNTER : DINT := 1;
   RES_B1_RECLOSE_OFF : BOOL;
   RES_B1_RECLOSE_TIMER : TIMER := (PRE := 1000);
   RES_B1_RECLOSED : BOOL;
   RES_B1_REQ_CLOSE : BOOL := 1;
   RES_B1_REQ_CONNECT : BOOL := 1;
   RES_B1_REQ_DISCONNECT : BOOL;
   RES_B1_REQ_OPEN : BOOL;
   RES_B1_REQ_RECLOSE : BOOL;
   RES_B1_SENSOR_ERROR : BOOL;
   RES_B1L1_CURRENT : REAL := 0.34258947;
   RES_B1L1_CURRENT_RAW : REAL := 5613.0;
   RES_B1L2_CURRENT : REAL := -0.001892085;
   RES_B1L2_CURRENT_RAW : REAL := -31.0;
   RES_B1L3_CURRENT : REAL := -0.0040893448;
   RES_B1L3_CURRENT_RAW : REAL := -67.0;
   RES_B1L4_CURRENT : REAL := -0.006164535;
   RES_B1L4_CURRENT_RAW : REAL := -101.0;
   RES_B1L5_CURRENT : REAL := 0.019348094;
   RES_B1L5_CURRENT_RAW : REAL := 317.0;
   RES_B2_CLOSE_PROXY : BOOL := 1;
   RES_B2_CLOSED : BOOL := 1;
   RES_B2_COMMAND_CHANGED : BOOL;
   RES_B2_COMMAND_CHANGED_TIMER : TIMER;
   RES_B2_CURRENT_CHECK : REAL := 0.0150756445;
   RES_B2_CURRENT_RAW : REAL := -1.0;
   RES_B2_DISCREPANCY : REAL := 0.015686015;
   RES_B2_FAULT : BOOL;
   RES_B2_FAULT_CANCEL : BOOL := 1;
   RES_B2_FAULT_PENDING : BOOL;
   RES_B2_FAULT_REQ : BOOL;
   RES_B2_FAULT_RETHROW_TIMER : TIMER := (PRE := 100);
   RES_B2_FAULT_TRIP : BOOL;
   RES_B2_INT_REQ_CLOSE : BOOL := 1;
   RES_B2_INT_REQ_CONNECT : BOOL := 1;
   RES_B2_MISMATCH : BOOL;
   RES_B2_NEW_FAULT : BOOL;
   RES_B2_RECLOSE_COUNTER : DINT := 3;
   RES_B2_RECLOSE_OFF : BOOL;
   RES_B2_RECLOSE_TIMER : TIMER := (PRE := 1000);
   RES_B2_RECLOSED : BOOL;
   RES_B2_REQ_CLOSE : BOOL := 1;
   RES_B2_REQ_CONNECT : BOOL := 1;
   RES_B2_REQ_DISCONNECT : BOOL;
   RES_B2_REQ_OPEN : BOOL;
   RES_B2_REQ_RECLOSE : BOOL;
   RES_B2_SENSOR_ERROR : BOOL;
   RES_B2L1_CURRENT : REAL := 0.00695799;
   RES_B2L1_CURRENT_RAW : REAL := 114.0;
   RES_B2L2_CURRENT : REAL := 0.00622557;
   RES_B2L2_CURRENT_RAW : REAL := 102.0;
   RES_B2L3_CURRENT : REAL;
   RES_B2L3_CURRENT_RAW : REAL := 0.004211415;
   RES_B2L4_CURRENT : REAL := -0.000427245;
   RES_B2L4_CURRENT_RAW : REAL := -7.0;
   RES_B2L5_CURRENT : REAL := 0.00231933;
   RES_B2L5_CURRENT_RAW : REAL := 38.0;
   RES_B3_CLOSE_PROXY : BOOL;
   RES_B3_CLOSED : BOOL;
   RES_B3_COMMAND_CHANGED : BOOL;
   RES_B3_COMMAND_CHANGED_TIMER : TIMER;
   RES_B3_CURRENT_CHECK : REAL := 0.016967729;
   RES_B3_CURRENT_RAW : REAL := -1.0;
   RES_B3_DISCREPANCY : REAL := 0.017578099;
   RES_B3_FAULT : BOOL;
   RES_B3_FAULT_CANCEL : BOOL;
   RES_B3_FAULT_PENDING : BOOL := 1;
   RES_B3_FAULT_REQ : BOOL := 1;
   RES_B3_FAULT_RETHROW_TIMER : TIMER := (PRE := 100);
   RES_B3_FAULT_TRIP : BOOL := 1;
   RES_B3_INT_REQ_CLOSE : BOOL;
   RES_B3_INT_REQ_CONNECT : BOOL;
   RES_B3_MISMATCH : BOOL;
   RES_B3_NEW_FAULT : BOOL;
   RES_B3_RECLOSE_COUNTER : DINT := 4;
   RES_B3_RECLOSE_OFF : BOOL := 1;
   RES_B3_RECLOSE_TIMER : TIMER := (PRE := 1000);
   RES_B3_RECLOSED : BOOL;
   RES_B3_REQ_CLOSE : BOOL;
   RES_B3_REQ_CONNECT : BOOL;
   RES_B3_REQ_DISCONNECT : BOOL := 1;
   RES_B3_REQ_OPEN : BOOL := 1;
   RES_B3_REQ_RECLOSE : BOOL;
   RES_B3_SENSOR_ERROR : BOOL;
   RES_B3L1_CURRENT : REAL := 0.00390624;
   RES_B3L1_CURRENT_RAW : REAL := 64.0;
   RES_B3L2_CURRENT : REAL := 0.00500487;
   RES_B3L2_CURRENT_RAW : REAL := 82.0;
   RES_B3L3_CURRENT : REAL := -0.00292968;
   RES_B3L3_CURRENT_RAW : REAL := -48.0;
   RES_B3L4_CURRENT : REAL := 0.00256347;
   RES_B3L4_CURRENT_RAW : REAL := 42.0;
   RES_B3L5_CURRENT : REAL := 0.00842283;
   RES_B3L5_CURRENT_RAW : REAL := 138.0;
   RES_B4_CLOSE_PROXY : BOOL := 1;
   RES_B4_CLOSED : BOOL := 1;
   RES_B4_COMMAND_CHANGED : BOOL;
   RES_B4_COMMAND_CHANGED_TIMER : TIMER;
   RES_B4_CURRENT_CHECK : REAL := 0.00598143;
   RES_B4_CURRENT_RAW : REAL;
   RES_B4_DISCREPANCY : REAL := 0.00598143;
   RES_B4_FAULT : BOOL;
   RES_B4_FAULT_CANCEL : BOOL := 1;
   RES_B4_FAULT_PENDING : BOOL;
   RES_B4_FAULT_REQ : BOOL;
   RES_B4_FAULT_RETHROW_TIMER : TIMER := (PRE := 100);
   RES_B4_FAULT_TRIP : BOOL;
   RES_B4_INT_REQ_CLOSE : BOOL := 1;
   RES_B4_INT_REQ_CONNECT : BOOL := 1;
   RES_B4_MISMATCH : BOOL;
   RES_B4_NEW_FAULT : BOOL;
   RES_B4_RECLOSE_COUNTER : DINT := 2;
   RES_B4_RECLOSE_OFF : BOOL;
   RES_B4_RECLOSE_TIMER : TIMER := (PRE := 1000);
   RES_B4_RECLOSED : BOOL;
   RES_B4_REQ_CLOSE : BOOL := 1;
   RES_B4_REQ_CONNECT : BOOL := 1;
   RES_B4_REQ_DISCONNECT : BOOL;
   RES_B4_REQ_OPEN : BOOL;
   RES_B4_REQ_RECLOSE : BOOL;
   RES_B4_SENSOR_ERROR : BOOL;
   RES_B4L1_CURRENT : REAL := 0.001525875;
   RES_B4L1_CURRENT_RAW : REAL := 25.0;
   RES_B4L2_CURRENT : REAL := 0.0021362249;
   RES_B4L2_CURRENT_RAW : REAL := 35.0;
   RES_B4L3_CURRENT : REAL := -0.00170898;
   RES_B4L3_CURRENT_RAW : REAL := -28.0;
   RES_B4L4_CURRENT : REAL := 0.00402831;
   RES_B4L4_CURRENT_RAW : REAL := 66.0;
   RES_B4L5_CURRENT : REAL;
   RES_B4L5_CURRENT_RAW : REAL;
   RES_BUS1_CURRENT : REAL := 0.34241757;
   RES_BUS2_CURRENT : REAL := -0.00061037;
   RES_BUS3_CURRENT : REAL := -0.00061037;
   RES_BUS4_CURRENT : REAL;
   RES_BUS_FAULT_THRESHOLD : REAL := 0.2;
   RES_Deadband : REAL := 0.005;
   RES_HighVoltage : BOOL;
   RES_HighVoltageThreshold : REAL;
   RES_LowVoltage : BOOL;
   RES_LowVoltageThreshold : REAL;
   RES_MAIN_CLOSE_PROXY : BOOL := 1;
   RES_MAIN_CLOSED : BOOL := 1;
   RES_MAIN_COMMAND_CHANGED : BOOL;
   RES_MAIN_COMMAND_CHANGED_TIMER : TIMER;
   RES_MAIN_CURRENT : REAL := 0.14404732;
   RES_MAIN_CURRENT_CHECK : REAL := 0.3411968;
   RES_MAIN_CURRENT_RAW : REAL := 236.0;
   RES_MAIN_DISCREPANCY : REAL := 0.19714949;
   RES_MAIN_FAULT : BOOL;
   RES_MAIN_FAULT_CANCEL : BOOL := 1;
   RES_MAIN_FAULT_PENDING : BOOL;
   RES_MAIN_FAULT_REQ : BOOL;
   RES_MAIN_FAULT_RETHROW_TIMER : TIMER := (PRE := 100);
   RES_MAIN_FAULT_THRESHOLD : REAL := 4.0;
   RES_MAIN_FAULT_TRIP : BOOL;
   RES_MAIN_INT_REQ_CLOSE : BOOL := 1;
   RES_MAIN_INT_REQ_CONNECT : BOOL := 1;
   RES_MAIN_MISMATCH : BOOL;
   RES_MAIN_NEW_FAULT : BOOL;
   RES_MAIN_RECLOSE_COUNTER : DINT;
   RES_MAIN_RECLOSE_OFF : BOOL;
   RES_MAIN_RECLOSE_TIMER : TIMER := (PRE := 1000);
   RES_MAIN_RECLOSED : BOOL;
   RES_MAIN_REQ_CLOSE : BOOL := 1;
   RES_MAIN_REQ_CONNECT : BOOL := 1;
   RES_MAIN_REQ_DISCONNECT : BOOL;
   RES_MAIN_REQ_OPEN : BOOL;
   RES_MAIN_REQ_RECLOSE : BOOL;
   RES_MAIN_SENSOR_ERROR : BOOL;
   RES_MAIN_VOLTAGE : REAL := 7.0;
   RES_MAIN_VOLTAGE_RAW : REAL := 7.0;
   RESB1L1_CLOSE_PROXY : BOOL := 1;
   RESB1L1_CLOSE_RELAY : BOOL;
   RESB1L1_CLOSED : BOOL := 1;
   RESB1L1_CommandChanged : BOOL;
   RESB1L1_CommandChangedTimer : ALIAS FOR CL_TIMER00;
   RESB1L1_CONNECT_PROXY : BOOL;
   RESB1L1_ConnectFail : BOOL;
   RESB1L1_DisconnectFail : BOOL;
   RESB1L1_ForceConnect : BOOL;
   RESB1L1_INT_REQ_CLOSE : BOOL := 1;
   RESB1L1_INT_REQ_CONNECT : BOOL := 1;
   RESB1L1_OPEN : BOOL;
   RESB1L1_Price : REAL := 6.0;
   RESB1L1_PriceThreshold : REAL := 25.0;
   RESB1L1_REQ_CLOSE : BOOL := 1;
   RESB1L1_REQ_CONNECT : BOOL := 1;
   RESB1L1_REQ_DISCONNECT : BOOL;
   RESB1L1_REQ_OPEN : BOOL;
   RESB1L3CURR : REAL;
   RESB2L1_CLOSE_PROXY : BOOL := 1;
   RESB2L1_CLOSED : BOOL := 1;
   RESB2L1_CommandChanged : BOOL;
   RESB2L1_CommandChangedTimer : ALIAS FOR CL_TIMER00;
   RESB2L1_ConnectFail : BOOL;
   RESB2L1_DisconnectFail : BOOL;
   RESB2L1_ForceConnect : BOOL;
   RESB2L1_INT_REQ_CLOSE : BOOL := 1;
   RESB2L1_INT_REQ_CONNECT : BOOL := 1;
   RESB2L1_OPEN : BOOL;
   RESB2L1_Price : REAL := 6.0;
   RESB2L1_PriceThreshold : REAL := 25.0;
   RESB2L1_REQ_CLOSE : BOOL := 1;
   RESB2L1_REQ_CONNECT : BOOL := 1;
   RESB2L1_REQ_DISCONNECT : BOOL;
   RESB2L1_REQ_OPEN : BOOL;
   SF_CLOSE_PROXY : BOOL;
   SF_INT_REQ_CLOSE : BOOL;
   SF_INT_REQ_CONNECT : BOOL;
   SF_MAX_CURRENT : REAL;
   SF_POWER_AVAILABLE : BOOL;
   SF_REQ_CLOSE : BOOL;
   SF_REQ_CONNECT : BOOL;
   SF_REQ_DISCONNECT : BOOL;
   SF_REQ_OPEN : BOOL;
   VOLTAGE_SCALE : REAL := 1.0;
END_VAR

ROUTINE IMPORT_DATA   (* ladder *)
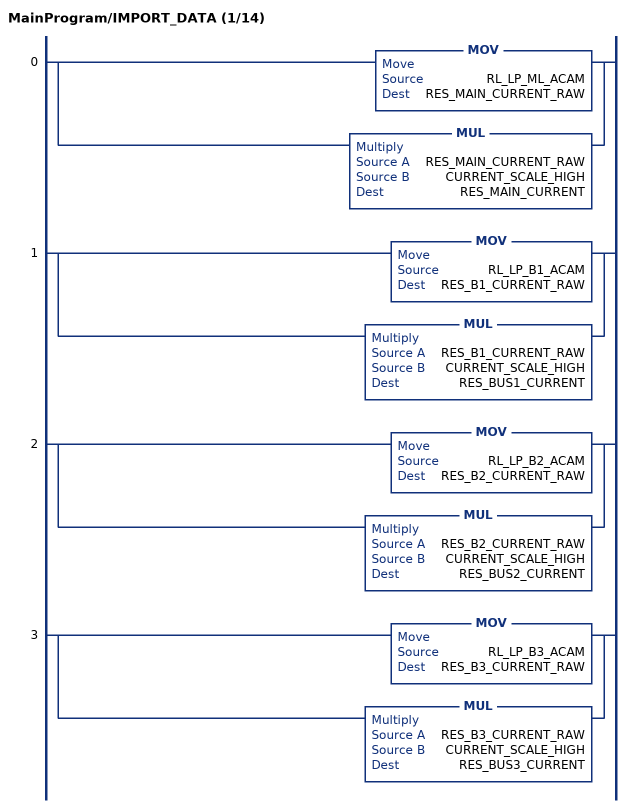
   0: [MOV(RL_LP_ML_ACAM,RES_MAIN_CURRENT_RAW) ,MUL(RES_MAIN_CURRENT_RAW,CURRENT_SCALE_HIGH,RES_MAIN_CURRENT) ];
   1: [MOV(RL_LP_B1_ACAM,RES_B1_CURRENT_RAW) ,MUL(RES_B1_CURRENT_RAW,CURRENT_SCALE_HIGH,RES_BUS1_CURRENT) ];
   2: [MOV(RL_LP_B2_ACAM,RES_B2_CURRENT_RAW) ,MUL(RES_B2_CURRENT_RAW,CURRENT_SCALE_HIGH,RES_BUS2_CURRENT) ];
   3: [MOV(RL_LP_B3_ACAM,RES_B3_CURRENT_RAW) ,MUL(RES_B3_CURRENT_RAW,CURRENT_SCALE_HIGH,RES_BUS3_CURRENT) ];
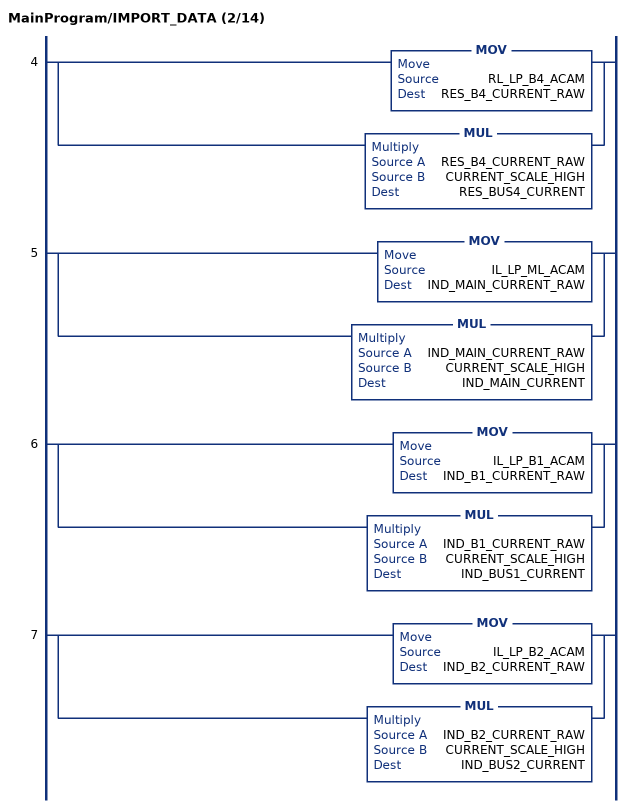
   4: [MOV(RL_LP_B4_ACAM,RES_B4_CURRENT_RAW) ,MUL(RES_B4_CURRENT_RAW,CURRENT_SCALE_HIGH,RES_BUS4_CURRENT) ];
   5: [MOV(IL_LP_ML_ACAM,IND_MAIN_CURRENT_RAW) ,MUL(IND_MAIN_CURRENT_RAW,CURRENT_SCALE_HIGH,IND_MAIN_CURRENT) ];
   6: [MOV(IL_LP_B1_ACAM,IND_B1_CURRENT_RAW) ,MUL(IND_B1_CURRENT_RAW,CURRENT_SCALE_HIGH,IND_BUS1_CURRENT) ];
   7: [MOV(IL_LP_B2_ACAM,IND_B2_CURRENT_RAW) ,MUL(IND_B2_CURRENT_RAW,CURRENT_SCALE_HIGH,IND_BUS2_CURRENT) ];
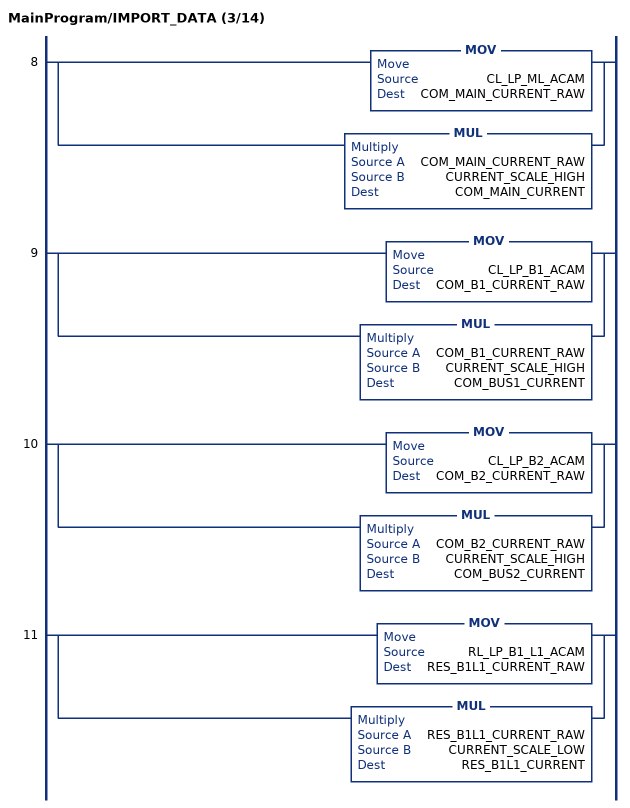
   8: [MOV(CL_LP_ML_ACAM,COM_MAIN_CURRENT_RAW) ,MUL(COM_MAIN_CURRENT_RAW,CURRENT_SCALE_HIGH,COM_MAIN_CURRENT) ];
   9: [MOV(CL_LP_B1_ACAM,COM_B1_CURRENT_RAW) ,MUL(COM_B1_CURRENT_RAW,CURRENT_SCALE_HIGH,COM_BUS1_CURRENT) ];
   10: [MOV(CL_LP_B2_ACAM,COM_B2_CURRENT_RAW) ,MUL(COM_B2_CURRENT_RAW,CURRENT_SCALE_HIGH,COM_BUS2_CURRENT) ];
   11: [MOV(RL_LP_B1_L1_ACAM,RES_B1L1_CURRENT_RAW) ,MUL(RES_B1L1_CURRENT_RAW,CURRENT_SCALE_LOW,RES_B1L1_CURRENT) ];
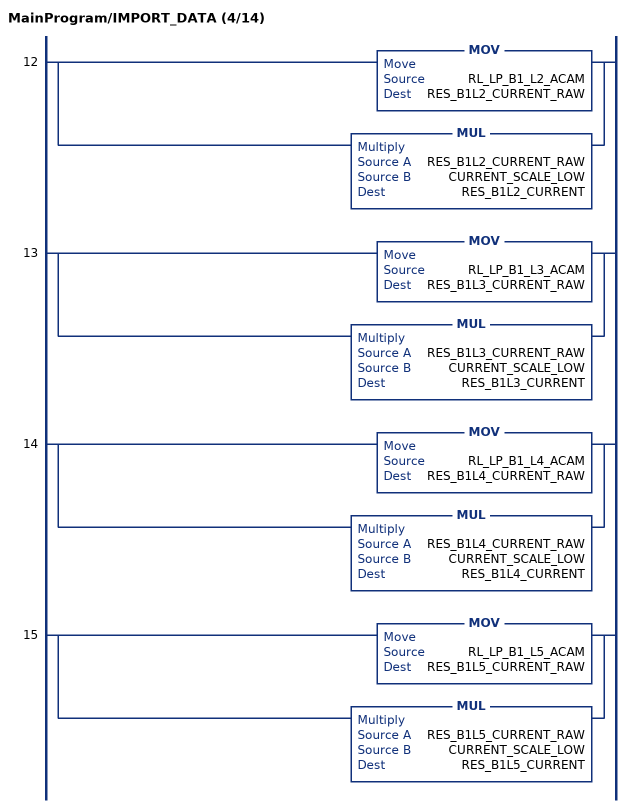
   12: [MOV(RL_LP_B1_L2_ACAM,RES_B1L2_CURRENT_RAW) ,MUL(RES_B1L2_CURRENT_RAW,CURRENT_SCALE_LOW,RES_B1L2_CURRENT) ];
   13: [MOV(RL_LP_B1_L3_ACAM,RES_B1L3_CURRENT_RAW) ,MUL(RES_B1L3_CURRENT_RAW,CURRENT_SCALE_LOW,RES_B1L3_CURRENT) ];
   14: [MOV(RL_LP_B1_L4_ACAM,RES_B1L4_CURRENT_RAW) ,MUL(RES_B1L4_CURRENT_RAW,CURRENT_SCALE_LOW,RES_B1L4_CURRENT) ];
   15: [MOV(RL_LP_B1_L5_ACAM,RES_B1L5_CURRENT_RAW) ,MUL(RES_B1L5_CURRENT_RAW,CURRENT_SCALE_LOW,RES_B1L5_CURRENT) ];
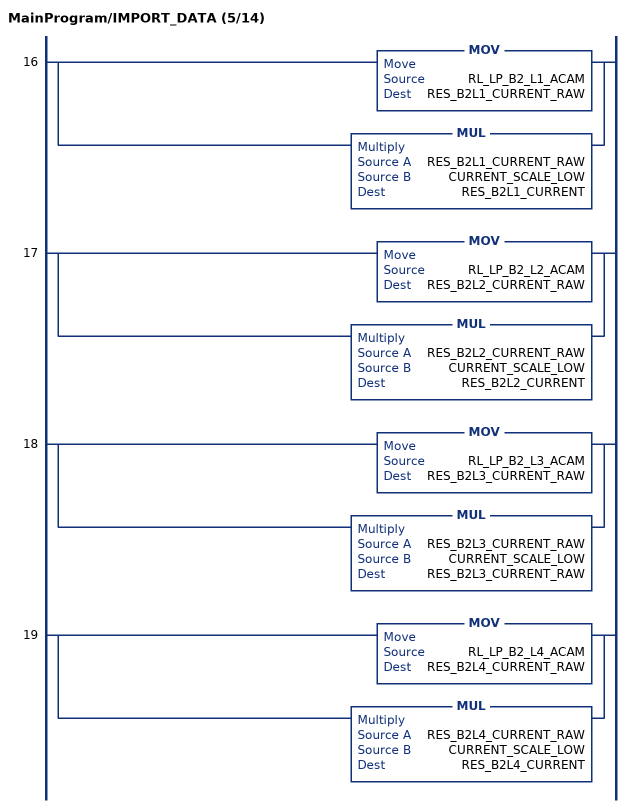
   16: [MOV(RL_LP_B2_L1_ACAM,RES_B2L1_CURRENT_RAW) ,MUL(RES_B2L1_CURRENT_RAW,CURRENT_SCALE_LOW,RES_B2L1_CURRENT) ];
   17: [MOV(RL_LP_B2_L2_ACAM,RES_B2L2_CURRENT_RAW) ,MUL(RES_B2L2_CURRENT_RAW,CURRENT_SCALE_LOW,RES_B2L2_CURRENT) ];
   18: [MOV(RL_LP_B2_L3_ACAM,RES_B2L3_CURRENT_RAW) ,MUL(RES_B2L3_CURRENT_RAW,CURRENT_SCALE_LOW,RES_B2L3_CURRENT_RAW) ];
   19: [MOV(RL_LP_B2_L4_ACAM,RES_B2L4_CURRENT_RAW) ,MUL(RES_B2L4_CURRENT_RAW,CURRENT_SCALE_LOW,RES_B2L4_CURRENT) ];
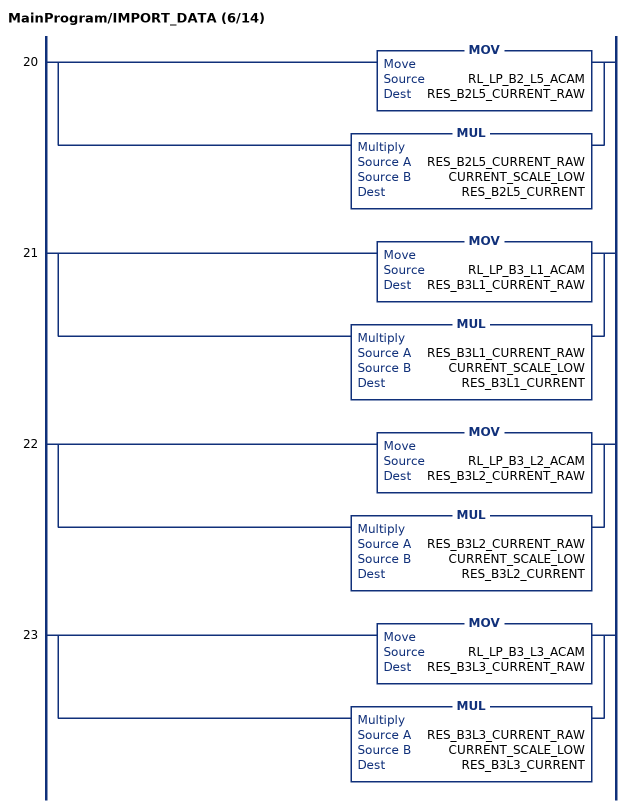
   20: [MOV(RL_LP_B2_L5_ACAM,RES_B2L5_CURRENT_RAW) ,MUL(RES_B2L5_CURRENT_RAW,CURRENT_SCALE_LOW,RES_B2L5_CURRENT) ];
   21: [MOV(RL_LP_B3_L1_ACAM,RES_B3L1_CURRENT_RAW) ,MUL(RES_B3L1_CURRENT_RAW,CURRENT_SCALE_LOW,RES_B3L1_CURRENT) ];
   22: [MOV(RL_LP_B3_L2_ACAM,RES_B3L2_CURRENT_RAW) ,MUL(RES_B3L2_CURRENT_RAW,CURRENT_SCALE_LOW,RES_B3L2_CURRENT) ];
   23: [MOV(RL_LP_B3_L3_ACAM,RES_B3L3_CURRENT_RAW) ,MUL(RES_B3L3_CURRENT_RAW,CURRENT_SCALE_LOW,RES_B3L3_CURRENT) ];
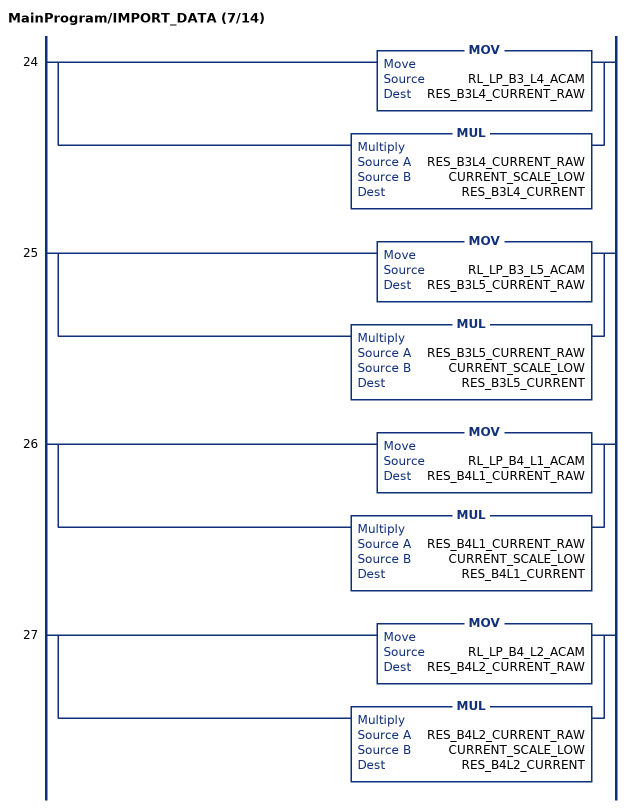
   24: [MOV(RL_LP_B3_L4_ACAM,RES_B3L4_CURRENT_RAW) ,MUL(RES_B3L4_CURRENT_RAW,CURRENT_SCALE_LOW,RES_B3L4_CURRENT) ];
   25: [MOV(RL_LP_B3_L5_ACAM,RES_B3L5_CURRENT_RAW) ,MUL(RES_B3L5_CURRENT_RAW,CURRENT_SCALE_LOW,RES_B3L5_CURRENT) ];
   26: [MOV(RL_LP_B4_L1_ACAM,RES_B4L1_CURRENT_RAW) ,MUL(RES_B4L1_CURRENT_RAW,CURRENT_SCALE_LOW,RES_B4L1_CURRENT) ];
   27: [MOV(RL_LP_B4_L2_ACAM,RES_B4L2_CURRENT_RAW) ,MUL(RES_B4L2_CURRENT_RAW,CURRENT_SCALE_LOW,RES_B4L2_CURRENT) ];
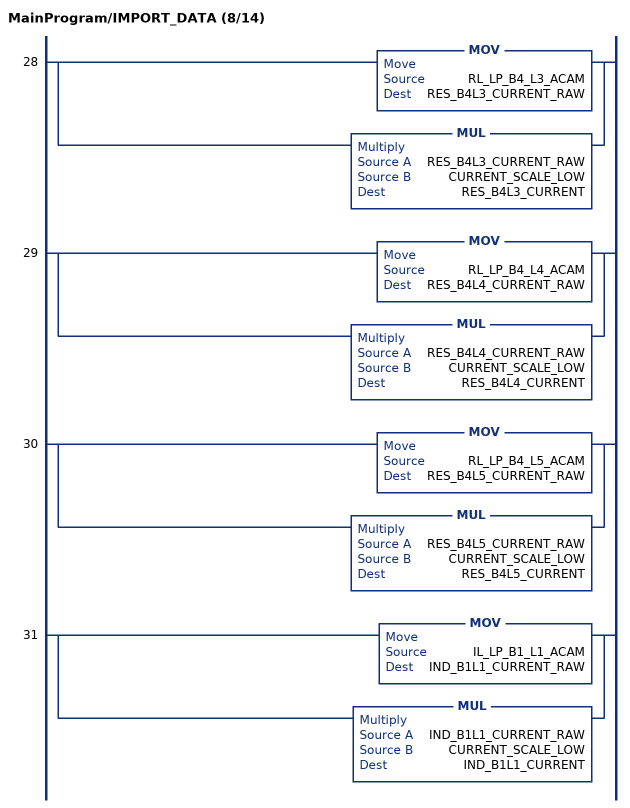
   28: [MOV(RL_LP_B4_L3_ACAM,RES_B4L3_CURRENT_RAW) ,MUL(RES_B4L3_CURRENT_RAW,CURRENT_SCALE_LOW,RES_B4L3_CURRENT) ];
   29: [MOV(RL_LP_B4_L4_ACAM,RES_B4L4_CURRENT_RAW) ,MUL(RES_B4L4_CURRENT_RAW,CURRENT_SCALE_LOW,RES_B4L4_CURRENT) ];
   30: [MOV(RL_LP_B4_L5_ACAM,RES_B4L5_CURRENT_RAW) ,MUL(RES_B4L5_CURRENT_RAW,CURRENT_SCALE_LOW,RES_B4L5_CURRENT) ];
   31: [MOV(IL_LP_B1_L1_ACAM,IND_B1L1_CURRENT_RAW) ,MUL(IND_B1L1_CURRENT_RAW,CURRENT_SCALE_LOW,IND_B1L1_CURRENT) ];
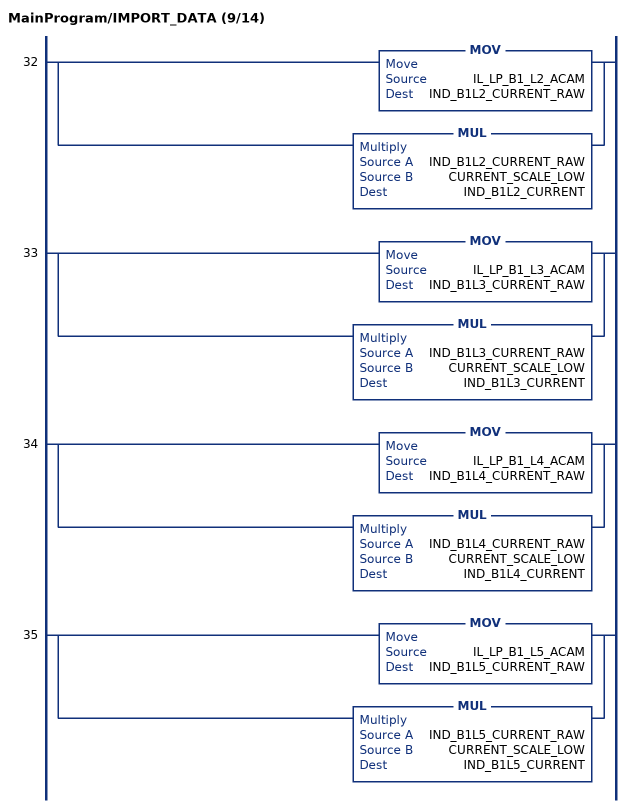
   32: [MOV(IL_LP_B1_L2_ACAM,IND_B1L2_CURRENT_RAW) ,MUL(IND_B1L2_CURRENT_RAW,CURRENT_SCALE_LOW,IND_B1L2_CURRENT) ];
   33: [MOV(IL_LP_B1_L3_ACAM,IND_B1L3_CURRENT_RAW) ,MUL(IND_B1L3_CURRENT_RAW,CURRENT_SCALE_LOW,IND_B1L3_CURRENT) ];
   34: [MOV(IL_LP_B1_L4_ACAM,IND_B1L4_CURRENT_RAW) ,MUL(IND_B1L4_CURRENT_RAW,CURRENT_SCALE_LOW,IND_B1L4_CURRENT) ];
   35: [MOV(IL_LP_B1_L5_ACAM,IND_B1L5_CURRENT_RAW) ,MUL(IND_B1L5_CURRENT_RAW,CURRENT_SCALE_LOW,IND_B1L5_CURRENT) ];
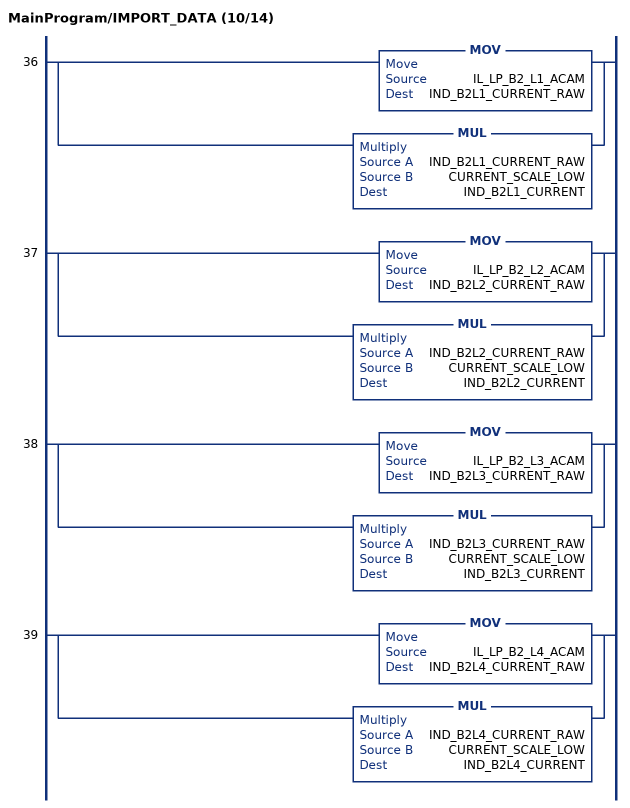
   36: [MOV(IL_LP_B2_L1_ACAM,IND_B2L1_CURRENT_RAW) ,MUL(IND_B2L1_CURRENT_RAW,CURRENT_SCALE_LOW,IND_B2L1_CURRENT) ];
   37: [MOV(IL_LP_B2_L2_ACAM,IND_B2L2_CURRENT_RAW) ,MUL(IND_B2L2_CURRENT_RAW,CURRENT_SCALE_LOW,IND_B2L2_CURRENT) ];
   38: [MOV(IL_LP_B2_L3_ACAM,IND_B2L3_CURRENT_RAW) ,MUL(IND_B2L3_CURRENT_RAW,CURRENT_SCALE_LOW,IND_B2L3_CURRENT) ];
   39: [MOV(IL_LP_B2_L4_ACAM,IND_B2L4_CURRENT_RAW) ,MUL(IND_B2L4_CURRENT_RAW,CURRENT_SCALE_LOW,IND_B2L4_CURRENT) ];
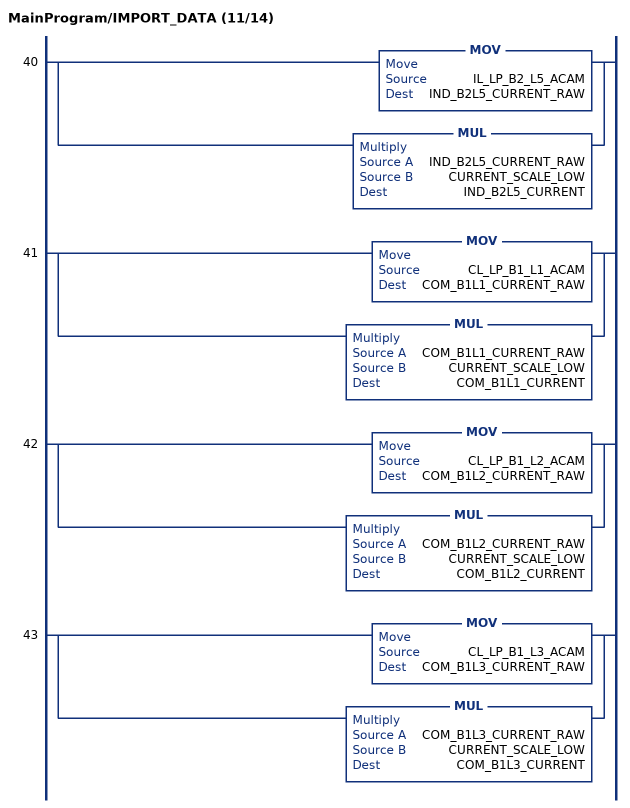
   40: [MOV(IL_LP_B2_L5_ACAM,IND_B2L5_CURRENT_RAW) ,MUL(IND_B2L5_CURRENT_RAW,CURRENT_SCALE_LOW,IND_B2L5_CURRENT) ];
   41: [MOV(CL_LP_B1_L1_ACAM,COM_B1L1_CURRENT_RAW) ,MUL(COM_B1L1_CURRENT_RAW,CURRENT_SCALE_LOW,COM_B1L1_CURRENT) ];
   42: [MOV(CL_LP_B1_L2_ACAM,COM_B1L2_CURRENT_RAW) ,MUL(COM_B1L2_CURRENT_RAW,CURRENT_SCALE_LOW,COM_B1L2_CURRENT) ];
   43: [MOV(CL_LP_B1_L3_ACAM,COM_B1L3_CURRENT_RAW) ,MUL(COM_B1L3_CURRENT_RAW,CURRENT_SCALE_LOW,COM_B1L3_CURRENT) ];
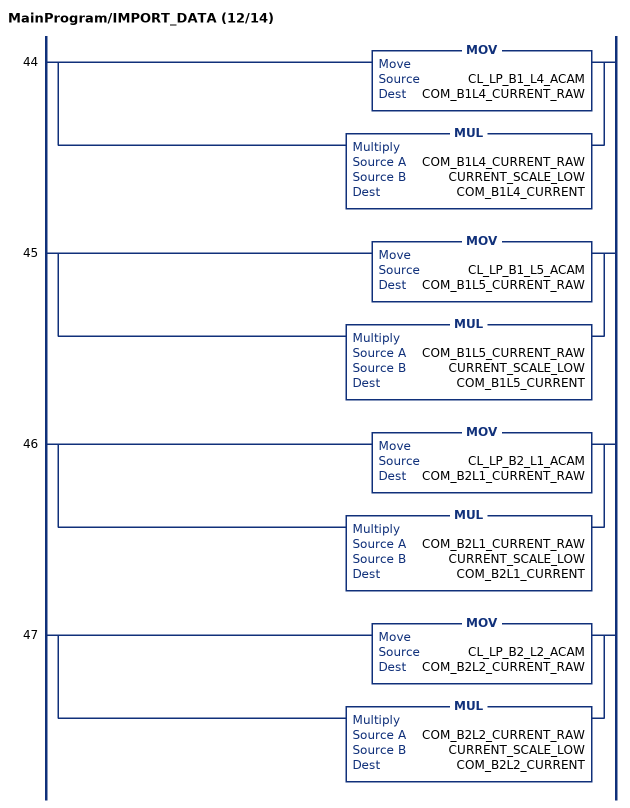
   44: [MOV(CL_LP_B1_L4_ACAM,COM_B1L4_CURRENT_RAW) ,MUL(COM_B1L4_CURRENT_RAW,CURRENT_SCALE_LOW,COM_B1L4_CURRENT) ];
   45: [MOV(CL_LP_B1_L5_ACAM,COM_B1L5_CURRENT_RAW) ,MUL(COM_B1L5_CURRENT_RAW,CURRENT_SCALE_LOW,COM_B1L5_CURRENT) ];
   46: [MOV(CL_LP_B2_L1_ACAM,COM_B2L1_CURRENT_RAW) ,MUL(COM_B2L1_CURRENT_RAW,CURRENT_SCALE_LOW,COM_B2L1_CURRENT) ];
   47: [MOV(CL_LP_B2_L2_ACAM,COM_B2L2_CURRENT_RAW) ,MUL(COM_B2L2_CURRENT_RAW,CURRENT_SCALE_LOW,COM_B2L2_CURRENT) ];
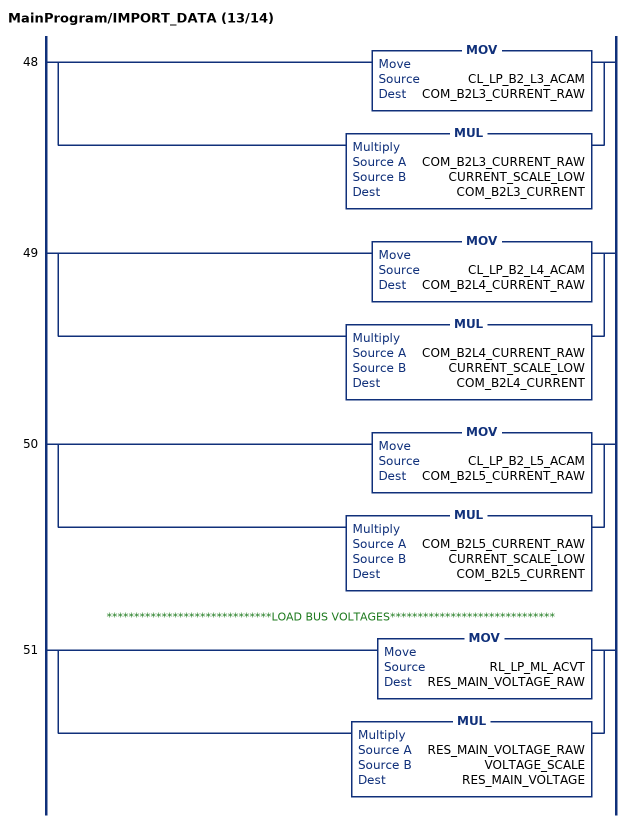
   48: [MOV(CL_LP_B2_L3_ACAM,COM_B2L3_CURRENT_RAW) ,MUL(COM_B2L3_CURRENT_RAW,CURRENT_SCALE_LOW,COM_B2L3_CURRENT) ];
   49: [MOV(CL_LP_B2_L4_ACAM,COM_B2L4_CURRENT_RAW) ,MUL(COM_B2L4_CURRENT_RAW,CURRENT_SCALE_LOW,COM_B2L4_CURRENT) ];
   50: [MOV(CL_LP_B2_L5_ACAM,COM_B2L5_CURRENT_RAW) ,MUL(COM_B2L5_CURRENT_RAW,CURRENT_SCALE_LOW,COM_B2L5_CURRENT) ];
   // ******************************LOAD BUS VOLTAGES******************************
   51: [MOV(RL_LP_ML_ACVT,RES_MAIN_VOLTAGE_RAW) ,MUL(RES_MAIN_VOLTAGE_RAW,VOLTAGE_SCALE,RES_MAIN_VOLTAGE) ];
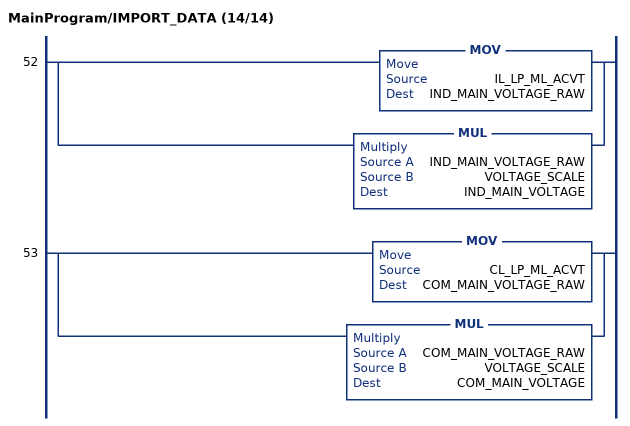
   52: [MOV(IL_LP_ML_ACVT,IND_MAIN_VOLTAGE_RAW) ,MUL(IND_MAIN_VOLTAGE_RAW,VOLTAGE_SCALE,IND_MAIN_VOLTAGE) ];
   53: [MOV(CL_LP_ML_ACVT,COM_MAIN_VOLTAGE_RAW) ,MUL(COM_MAIN_VOLTAGE_RAW,VOLTAGE_SCALE,COM_MAIN_VOLTAGE) ];
END_ROUTINE

ROUTINE MainRoutine   (* ladder *)
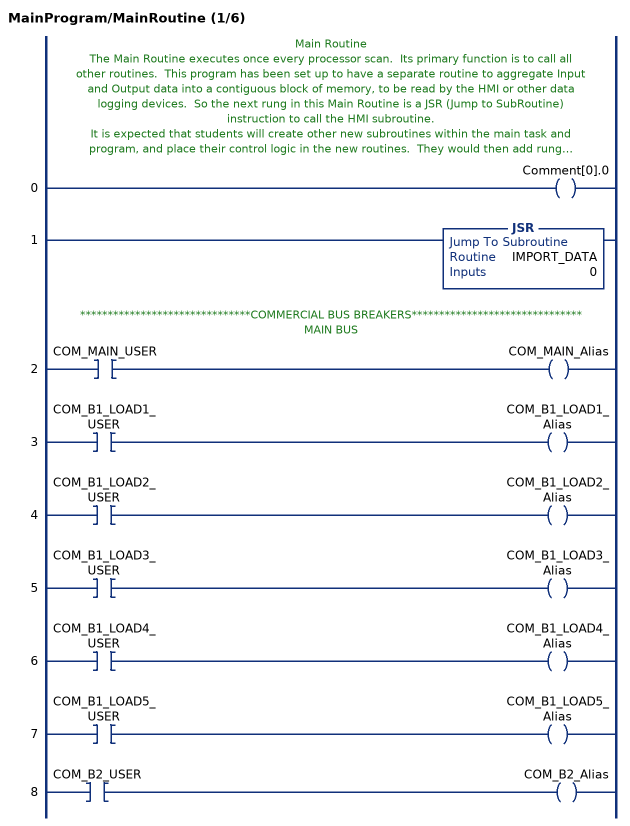
   // Main Routine
   // The Main Routine executes once every processor scan.  Its primary function is to call all other routines.  This program has been set up to have a separate routine to aggregate Input and Output data into a contiguous block of memory, to be read by the HMI or other data logging devices.  So the next rung in this Main Routine is a JSR (Jump to SubRoutine) instruction to call the HMI subroutine.
   // It is expected that students will create other new subroutines within the main task and program, and place their control logic in the new routines.  They would then add rungs within this Main Routine to call the new subroutines that contain their logic.
   0: OTE(Comment[0].0);
   1: JSR(IMPORT_DATA,0);
   // *******************************COMMERCIAL BUS BREAKERS*******************************
   // MAIN BUS
   2: XIC(COM_MAIN_USER)OTE(COM_MAIN_Alias);
   3: XIC(COM_B1_LOAD1_USER)OTE(COM_B1_LOAD1_Alias);
   4: XIC(COM_B1_LOAD2_USER)OTE(COM_B1_LOAD2_Alias);
   5: XIC(COM_B1_LOAD3_USER)OTE(COM_B1_LOAD3_Alias);
   6: XIC(COM_B1_LOAD4_USER)OTE(COM_B1_LOAD4_Alias);
   7: XIC(COM_B1_LOAD5_USER)OTE(COM_B1_LOAD5_Alias);
   8: XIC(COM_B2_USER)OTE(COM_B2_Alias);
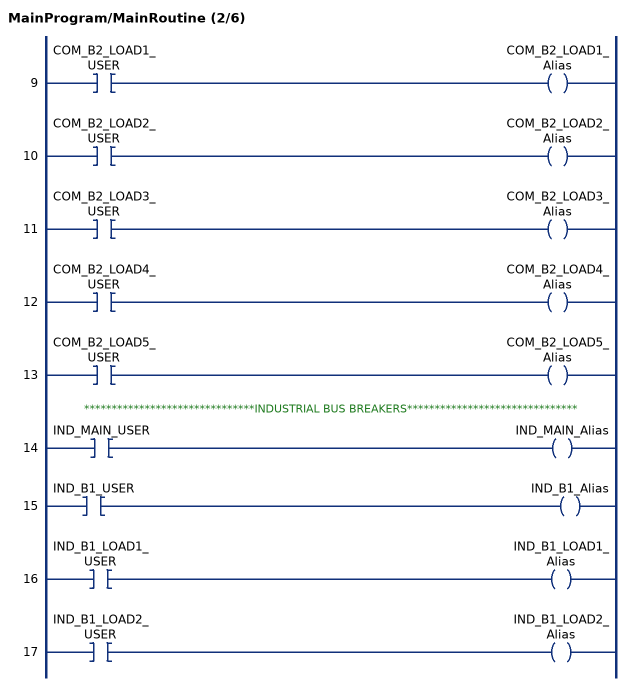
   9: XIC(COM_B2_LOAD1_USER)OTE(COM_B2_LOAD1_Alias);
   10: XIC(COM_B2_LOAD2_USER)OTE(COM_B2_LOAD2_Alias);
   11: XIC(COM_B2_LOAD3_USER)OTE(COM_B2_LOAD3_Alias);
   12: XIC(COM_B2_LOAD4_USER)OTE(COM_B2_LOAD4_Alias);
   13: XIC(COM_B2_LOAD5_USER)OTE(COM_B2_LOAD5_Alias);
   // *******************************INDUSTRIAL BUS BREAKERS*******************************
   14: XIC(IND_MAIN_USER)OTE(IND_MAIN_Alias);
   15: XIC(IND_B1_USER)OTE(IND_B1_Alias);
   16: XIC(IND_B1_LOAD1_USER)OTE(IND_B1_LOAD1_Alias);
   17: XIC(IND_B1_LOAD2_USER)OTE(IND_B1_LOAD2_Alias);
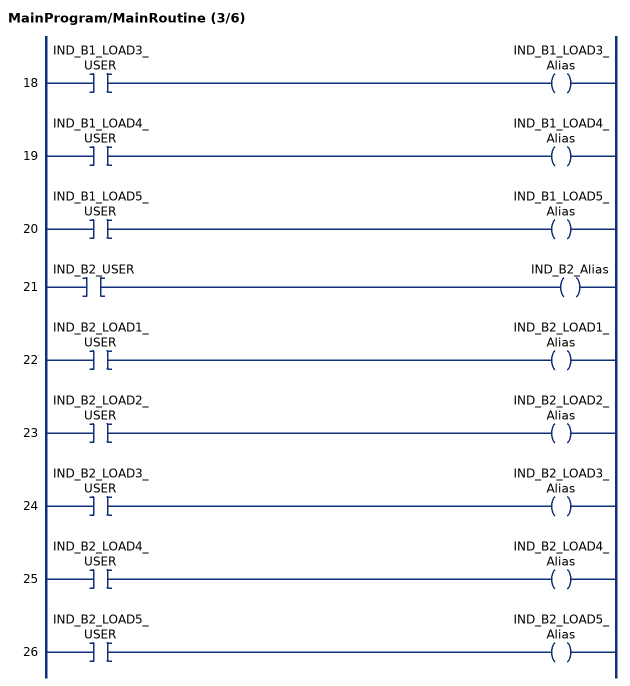
   18: XIC(IND_B1_LOAD3_USER)OTE(IND_B1_LOAD3_Alias);
   19: XIC(IND_B1_LOAD4_USER)OTE(IND_B1_LOAD4_Alias);
   20: XIC(IND_B1_LOAD5_USER)OTE(IND_B1_LOAD5_Alias);
   21: XIC(IND_B2_USER)OTE(IND_B2_Alias);
   22: XIC(IND_B2_LOAD1_USER)OTE(IND_B2_LOAD1_Alias);
   23: XIC(IND_B2_LOAD2_USER)OTE(IND_B2_LOAD2_Alias);
   24: XIC(IND_B2_LOAD3_USER)OTE(IND_B2_LOAD3_Alias);
   25: XIC(IND_B2_LOAD4_USER)OTE(IND_B2_LOAD4_Alias);
   26: XIC(IND_B2_LOAD5_USER)OTE(IND_B2_LOAD5_Alias);
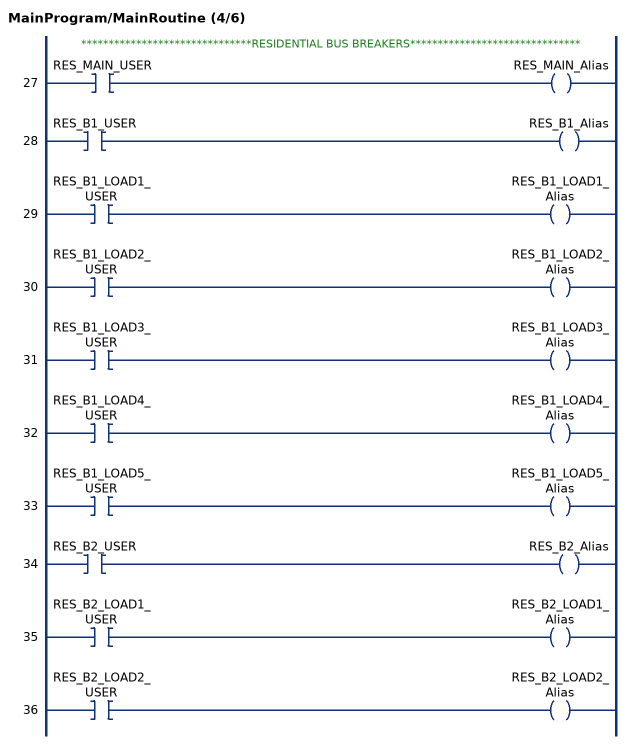
   // *******************************RESIDENTIAL BUS BREAKERS*******************************
   27: XIC(RES_MAIN_USER)OTE(RES_MAIN_Alias);
   28: XIC(RES_B1_USER)OTE(RES_B1_Alias);
   29: XIC(RES_B1_LOAD1_USER)OTE(RES_B1_LOAD1_Alias);
   30: XIC(RES_B1_LOAD2_USER)OTE(RES_B1_LOAD2_Alias);
   31: XIC(RES_B1_LOAD3_USER)OTE(RES_B1_LOAD3_Alias);
   32: XIC(RES_B1_LOAD4_USER)OTE(RES_B1_LOAD4_Alias);
   33: XIC(RES_B1_LOAD5_USER)OTE(RES_B1_LOAD5_Alias);
   34: XIC(RES_B2_USER)OTE(RES_B2_Alias);
   35: XIC(RES_B2_LOAD1_USER)OTE(RES_B2_LOAD1_Alias);
   36: XIC(RES_B2_LOAD2_USER)OTE(RES_B2_LOAD2_Alias);
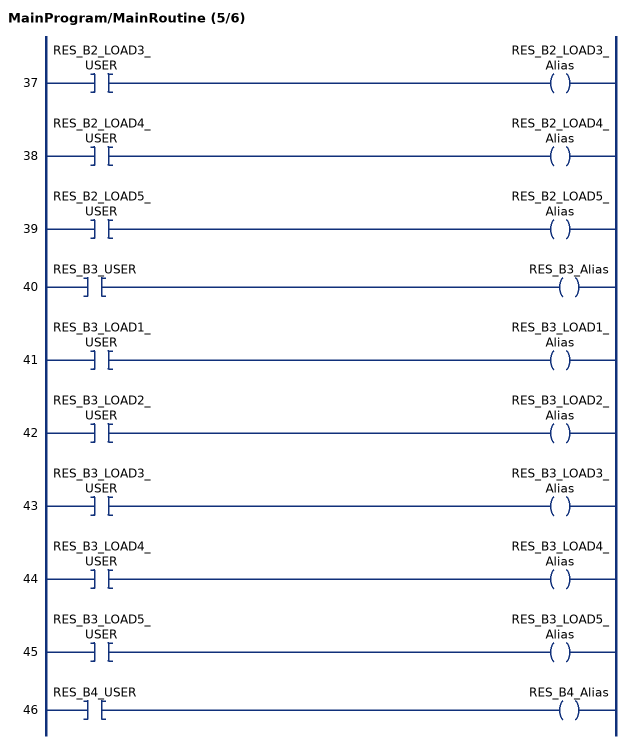
   37: XIC(RES_B2_LOAD3_USER)OTE(RES_B2_LOAD3_Alias);
   38: XIC(RES_B2_LOAD4_USER)OTE(RES_B2_LOAD4_Alias);
   39: XIC(RES_B2_LOAD5_USER)OTE(RES_B2_LOAD5_Alias);
   40: XIC(RES_B3_USER)OTE(RES_B3_Alias);
   41: XIC(RES_B3_LOAD1_USER)OTE(RES_B3_LOAD1_Alias);
   42: XIC(RES_B3_LOAD2_USER)OTE(RES_B3_LOAD2_Alias);
   43: XIC(RES_B3_LOAD3_USER)OTE(RES_B3_LOAD3_Alias);
   44: XIC(RES_B3_LOAD4_USER)OTE(RES_B3_LOAD4_Alias);
   45: XIC(RES_B3_LOAD5_USER)OTE(RES_B3_LOAD5_Alias);
   46: XIC(RES_B4_USER)OTE(RES_B4_Alias);
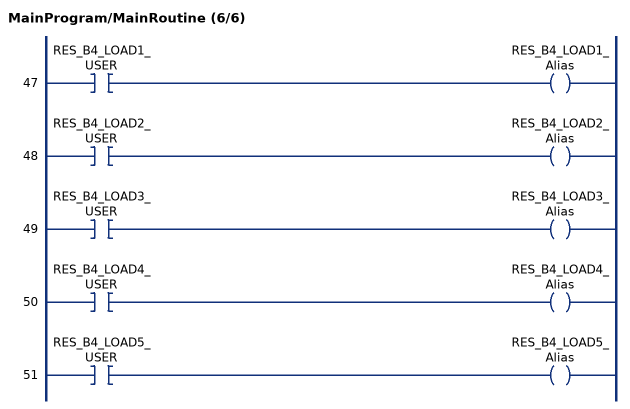
   47: XIC(RES_B4_LOAD1_USER)OTE(RES_B4_LOAD1_Alias);
   48: XIC(RES_B4_LOAD2_USER)OTE(RES_B4_LOAD2_Alias);
   49: XIC(RES_B4_LOAD3_USER)OTE(RES_B4_LOAD3_Alias);
   50: XIC(RES_B4_LOAD4_USER)OTE(RES_B4_LOAD4_Alias);
   51: XIC(RES_B4_LOAD5_USER)OTE(RES_B4_LOAD5_Alias);
END_ROUTINE
END_PROGRAM
